LIN {X 0,Y 487.933,Z 756.497,A -85,B 0,C 180,E1 -6477.523,E2 -6477.523} C_VEL
LIN {X 0,Y 487.892,Z 757.524,A -85,B 0,C 180,E1 -6478.349,E2 -6478.349} C_VEL
LIN {X 0,Y 487.819,Z 758.415,A -85,B 0,C 180,E1 -6480,E2 -6480} C_VEL
LIN {X 0,Y 487.834,Z 758.228,A -85,B 0,C 180,E1 -6480.825,E2 -6480.825} C_VEL
LIN {X 0,Y 487.892,Z 757.637,A -85,B 0,C 180,E1 -6481.651,E2 -6481.651} C_VEL
LIN {X 0,Y 487.933,Z 756.658,A -85,B 0,C 180,E1 -6482.477,E2 -6482.477} C_VEL
LIN {X 0,Y 487.977,Z 755.262,A -85,B 0,C 180,E1 -6483.303,E2 -6483.303} C_VEL
LIN {X 0,Y 487.984,Z 752.337,A -85,B 0,C 180,E1 -6484.543,E2 -6484.543} C_VEL
LIN {X 0,Y 488.159,Z 747.294,A -85,B 0,C 180,E1 -6486.059,E2 -6486.059} C_VEL
LIN {X 0,Y 488.271,Z 741.184,A -85,B 0,C 180,E1 -6487.443,E2 -6487.443} C_VEL
LIN {X 0,Y 488.524,Z 734.149,A -85,B 0,C 180,E1 -6488.688,E2 -6488.688} C_VEL
LIN {X 0,Y 488.845,Z 725.387,A -85,B 0,C 180,E1 -6489.934,E2 -6489.934} C_VEL
LIN {X 0,Y 489.125,Z 716.359,A -85,B 0,C 180,E1 -6490.975,E2 -6490.975} C_VEL
LIN {X 0,Y 489.537,Z 706.321,A -85,B 0,C 180,E1 -6491.91,E2 -6491.91} C_VEL
LIN {X 0,Y 489.887,Z 695.409,A -85,B 0,C 180,E1 -6492.732,E2 -6492.732} C_VEL
LIN {X 0,Y 490.166,Z 683.839,A -85,B 0,C 180,E1 -6493.421,E2 -6493.421} C_VEL
LIN {X 0,Y 490.537,Z 670.88,A -85,B 0,C 180,E1 -6493.991,E2 -6493.991} C_VEL
LIN {X 0,Y 490.801,Z 658.232,A -85,B 0,C 180,E1 -6494.38,E2 -6494.38} C_VEL
LIN {X 0,Y 490.962,Z 638.871,A -85,B 0,C 180,E1 -6494.72,E2 -6494.72} C_VEL
LIN {X 0,Y 491.66,Z 557.51,A -85,B 0,C 180,E1 -6496.021,E2 -6496.021} C_VEL
LIN {X 0,Y 489.823,Z 546.055,A -85,B 0,C 180,E1 -6496.292,E2 -6496.292} C_VEL
LIN {X 0,Y 490.318,Z 525.468,A -85,B 0,C 180,E1 -6499.249,E2 -6499.249} C_VEL
LIN {X 0,Y 490.759,Z 505.581,A -85,B 0,C 180,E1 -6502.081,E2 -6502.081} C_VEL
LIN {X 0,Y 491.164,Z 488.188,A -85,B 0,C 180,E1 -6504.517,E2 -6504.517} C_VEL
LIN {X 0,Y 490.28,Z 481.713,A -85,B 0,C 180,E1 -6505.47,E2 -6505.47} C_VEL
LIN {X 0,Y 488.805,Z 474.727,A -85,B 0,C 180,E1 -6506.545,E2 -6506.545} C_VEL
LIN {X 0,Y 488.726,Z 474.734,A -85,B 0,C 180,E1 -6509.27,E2 -6509.27} C_VEL
LIN {X 0,Y 488.705,Z 474.737,A -85,B 0,C 180,E1 -6512.147,E2 -6512.147} C_VEL
LIN {X 0,Y 488.72,Z 474.734,A -85,B 0,C 180,E1 -6515.115,E2 -6515.115} C_VEL
LIN {X 0,Y 488.683,Z 474.738,A -85,B 0,C 180,E1 -6518.2,E2 -6518.2} C_VEL
LIN {X 0,Y 488.72,Z 474.734,A -85,B 0,C 180,E1 -6520.345,E2 -6520.345} C_VEL
LIN {X 0,Y 488.688,Z 474.733,A -85,B 0,C 180,E1 -6523.654,E2 -6523.654} C_VEL
LIN {X 0,Y 488.695,Z 474.738,A -85,B 0,C 180,E1 -6526.346,E2 -6526.346} C_VEL
LIN {X 0,Y 488.721,Z 474.734,A -85,B 0,C 180,E1 -6528.586,E2 -6528.586} C_VEL
LIN {X 0,Y 488.682,Z 474.736,A -85,B 0,C 180,E1 -6531.8,E2 -6531.8} C_VEL
LIN {X 0,Y 488.73,Z 474.73,A -85,B 0,C 180,E1 -6535.052,E2 -6535.052} C_VEL
LIN {X 0,Y 488.709,Z 474.735,A -85,B 0,C 180,E1 -6538.045,E2 -6538.045} C_VEL
LIN {X 0,Y 488.735,Z 474.733,A -85,B 0,C 180,E1 -6540.73,E2 -6540.73} C_VEL
LIN {X 0,Y 488.818,Z 474.835,A -85,B 0,C 180,E1 -6543.323,E2 -6543.323} C_VEL
LIN {X 0,Y 492.279,Z 490.053,A -85,B 0,C 180,E1 -6545.701,E2 -6545.701} C_VEL
LIN {X 0,Y 491.607,Z 506.366,A -85,B 0,C 180,E1 -6547.959,E2 -6547.959} C_VEL
LIN {X 0,Y 490.829,Z 524.604,A -85,B 0,C 180,E1 -6550.446,E2 -6550.446} C_VEL
LIN {X 0,Y 493.202,Z 539.821,A -85,B 0,C 180,E1 -6550.788,E2 -6550.788} C_VEL
LIN {X 0,Y 491.994,Z 662.426,A -85,B 0,C 180,E1 -6552.691,E2 -6552.691} C_VEL
LIN {X 0,Y 491.67,Z 676.703,A -85,B 0,C 180,E1 -6553.076,E2 -6553.076} C_VEL
LIN {X 0,Y 491.321,Z 691.164,A -85,B 0,C 180,E1 -6553.649,E2 -6553.649} C_VEL
LIN {X 0,Y 490.845,Z 703.923,A -85,B 0,C 180,E1 -6554.32,E2 -6554.32} C_VEL
LIN {X 0,Y 490.282,Z 716.464,A -85,B 0,C 180,E1 -6555.153,E2 -6555.153} C_VEL
LIN {X 0,Y 489.827,Z 727.924,A -85,B 0,C 180,E1 -6556.094,E2 -6556.094} C_VEL
LIN {X 0,Y 489.367,Z 738.441,A -85,B 0,C 180,E1 -6557.138,E2 -6557.138} C_VEL
LIN {X 0,Y 488.945,Z 748.885,A -85,B 0,C 180,E1 -6558.391,E2 -6558.391} C_VEL
LIN {X 0,Y 488.603,Z 757.487,A -85,B 0,C 180,E1 -6559.642,E2 -6559.642} C_VEL
LIN {X 0,Y 488.314,Z 765.679,A -85,B 0,C 180,E1 -6561.1,E2 -6561.1} C_VEL
LIN {X 0,Y 488.084,Z 772.266,A -85,B 0,C 180,E1 -6562.554,E2 -6562.554} C_VEL
LIN {X 0,Y 488.017,Z 776.821,A -85,B 0,C 180,E1 -6563.797,E2 -6563.797} C_VEL
LIN {X 0,Y 487.962,Z 780.398,A -85,B 0,C 180,E1 -6565.043,E2 -6565.043} C_VEL
LIN {X 0,Y 487.955,Z 783.88,A -85,B 0,C 180,E1 -6566.697,E2 -6566.697} C_VEL
LIN {X 0,Y 487.887,Z 785.935,A -85,B 0,C 180,E1 -6568.349,E2 -6568.349} C_VEL
LIN {X 0,Y 487.817,Z 786.61,A -85,B 0,C 180,E1 -6570,E2 -6570} C_VEL
LIN {X 0,Y 487.887,Z 785.914,A -85,B 0,C 180,E1 -6571.651,E2 -6571.651} C_VEL
LIN {X 0,Y 487.955,Z 783.837,A -85,B 0,C 180,E1 -6573.303,E2 -6573.303} C_VEL
LIN {X 0,Y 487.962,Z 780.328,A -85,B 0,C 180,E1 -6574.958,E2 -6574.958} C_VEL
LIN {X 0,Y 488.027,Z 775.834,A -85,B 0,C 180,E1 -6576.456,E2 -6576.456} C_VEL
LIN {X 0,Y 488.151,Z 770.373,A -85,B 0,C 180,E1 -6577.861,E2 -6577.861} C_VEL
LIN {X 0,Y 488.396,Z 763.274,A -85,B 0,C 180,E1 -6579.317,E2 -6579.317} C_VEL
LIN {X 0,Y 488.709,Z 754.438,A -85,B 0,C 180,E1 -6580.775,E2 -6580.775} C_VEL
LIN {X 0,Y 489.084,Z 744.365,A -85,B 0,C 180,E1 -6582.128,E2 -6582.128} C_VEL
LIN {X 0,Y 489.532,Z 732.81,A -85,B 0,C 180,E1 -6583.385,E2 -6583.385} C_VEL
LIN {X 0,Y 490.01,Z 721.006,A -85,B 0,C 180,E1 -6584.43,E2 -6584.43} C_VEL
LIN {X 0,Y 490.577,Z 707.861,A -85,B 0,C 180,E1 -6585.369,E2 -6585.369} C_VEL
LIN {X 0,Y 491.05,Z 694.161,A -85,B 0,C 180,E1 -6586.139,E2 -6586.139} C_VEL
LIN {X 0,Y 491.481,Z 679.477,A -85,B 0,C 180,E1 -6586.752,E2 -6586.752} C_VEL
LIN {X 0,Y 491.806,Z 666.25,A -85,B 0,C 180,E1 -6587.142,E2 -6587.142} C_VEL
LIN {X 0,Y 492.03,Z 648.794,A -85,B 0,C 180,E1 -6587.455,E2 -6587.455} C_VEL
LIN {X 0,Y 493.022,Z 539.589,A -85,B 0,C 180,E1 -6589.157,E2 -6589.157} C_VEL
LIN {X 0,Y 490.811,Z 525.078,A -85,B 0,C 180,E1 -6589.491,E2 -6589.491} C_VEL
LIN {X 0,Y 492.007,Z 500.536,A -85,B 0,C 180,E1 -6592.908,E2 -6592.908} C_VEL
LIN {X 0,Y 492.543,Z 491.86,A -85,B 0,C 180,E1 -6594.152,E2 -6594.152} C_VEL
LIN {X 0,Y 491.719,Z 486.921,A -85,B 0,C 180,E1 -6594.938,E2 -6594.938} C_VEL
LIN {X 0,Y 489.179,Z 476.31,A -85,B 0,C 180,E1 -6596.751,E2 -6596.751} C_VEL
LIN {X 0,Y 488.79,Z 474.727,A -85,B 0,C 180,E1 -6597.058,E2 -6597.058} C_VEL
LIN {X 0,Y 488.713,Z 474.736,A -85,B 0,C 180,E1 -6600.363,E2 -6600.363} C_VEL
LIN {X 0,Y 488.737,Z 474.734,A -85,B 0,C 180,E1 -6603.484,E2 -6603.484} C_VEL
LIN {X 0,Y 488.684,Z 474.737,A -85,B 0,C 180,E1 -6606.355,E2 -6606.355} C_VEL
LIN {X 0,Y 488.703,Z 474.738,A -85,B 0,C 180,E1 -6609.254,E2 -6609.254} C_VEL
LIN {X 0,Y 488.726,Z 474.733,A -85,B 0,C 180,E1 -6611.602,E2 -6611.602} C_VEL
LIN {X 0,Y 488.715,Z 474.734,A -85,B 0,C 180,E1 -6614.801,E2 -6614.801} C_VEL
LIN {X 0,Y 488.694,Z 474.736,A -85,B 0,C 180,E1 -6617.475,E2 -6617.475} C_VEL
LIN {X 0,Y 488.736,Z 474.73,A -85,B 0,C 180,E1 -6619.677,E2 -6619.677} C_VEL
LIN {X 0,Y 488.683,Z 474.741,A -85,B 0,C 180,E1 -6622.841,E2 -6622.841} C_VEL
LIN {X 0,Y 488.736,Z 474.731,A -85,B 0,C 180,E1 -6625.888,E2 -6625.888} C_VEL
LIN {X 0,Y 488.697,Z 474.74,A -85,B 0,C 180,E1 -6628.821,E2 -6628.821} C_VEL
LIN {X 0,Y 488.749,Z 474.735,A -85,B 0,C 180,E1 -6631.671,E2 -6631.671} C_VEL
LIN {X 0,Y 488.806,Z 474.846,A -85,B 0,C 180,E1 -6633.646,E2 -6633.646} C_VEL
LIN {X 0,Y 491.471,Z 486.878,A -85,B 0,C 180,E1 -6635.912,E2 -6635.912} C_VEL
LIN {X 0,Y 491.925,Z 491.046,A -85,B 0,C 180,E1 -6636.643,E2 -6636.643} C_VEL
LIN {X 0,Y 490.778,Z 512.524,A -85,B 0,C 180,E1 -6640.117,E2 -6640.117} C_VEL
LIN {X 0,Y 490.085,Z 530.15,A -85,B 0,C 180,E1 -6642.904,E2 -6642.904} C_VEL
LIN {X 0,Y 489.754,Z 540.863,A -85,B 0,C 180,E1 -6644.578,E2 -6644.578} C_VEL
LIN {X 0,Y 492.036,Z 554.998,A -85,B 0,C 180,E1 -6644.916,E2 -6644.916} C_VEL
LIN {X 0,Y 490.94,Z 653.001,A -85,B 0,C 180,E1 -6646.575,E2 -6646.575} C_VEL
LIN {X 0,Y 490.687,Z 666.595,A -85,B 0,C 180,E1 -6646.98,E2 -6646.98} C_VEL
LIN {X 0,Y 490.427,Z 679.005,A -85,B 0,C 180,E1 -6647.52,E2 -6647.52} C_VEL
LIN {X 0,Y 490.086,Z 690.877,A -85,B 0,C 180,E1 -6648.209,E2 -6648.209} C_VEL
LIN {X 0,Y 489.611,Z 702.158,A -85,B 0,C 180,E1 -6649.036,E2 -6649.036} C_VEL
LIN {X 0,Y 489.215,Z 712.339,A -85,B 0,C 180,E1 -6649.969,E2 -6649.969} C_VEL
LIN {X 0,Y 488.877,Z 722.337,A -85,B 0,C 180,E1 -6651.11,E2 -6651.11} C_VEL
LIN {X 0,Y 488.51,Z 731.141,A -85,B 0,C 180,E1 -6652.353,E2 -6652.353} C_VEL
LIN {X 0,Y 488.403,Z 738.144,A -85,B 0,C 180,E1 -6653.597,E2 -6653.597} C_VEL
LIN {X 0,Y 488.04,Z 744.561,A -85,B 0,C 180,E1 -6655.043,E2 -6655.043} C_VEL
LIN {X 0,Y 488.059,Z 748.762,A -85,B 0,C 180,E1 -6656.285,E2 -6656.285} C_VEL
LIN {X 0,Y 487.993,Z 751.895,A -85,B 0,C 180,E1 -6657.524,E2 -6657.524} C_VEL
LIN {X 0,Y 487.899,Z 753.453,A -85,B 0,C 180,E1 -6658.349,E2 -6658.349} C_VEL
LIN {X 0,Y 487.835,Z 754.563,A -85,B 0,C 180,E1 -6659.175,E2 -6659.175} C_VEL
LIN {X 0,Y 487.834,Z 755.556,A -85,B 0,C 180,E1 -6660.825,E2 -6660.825} C_VEL
LIN {X 0,Y 487.892,Z 755.467,A -85,B 0,C 180,E1 -6661.651,E2 -6661.651} C_VEL
LIN {X 0,Y 487.93,Z 754.951,A -85,B 0,C 180,E1 -6662.477,E2 -6662.477} C_VEL
LIN {X 0,Y 487.963,Z 754.02,A -85,B 0,C 180,E1 -6663.303,E2 -6663.303} C_VEL
LIN {X 0,Y 487.965,Z 752.694,A -85,B 0,C 180,E1 -6664.13,E2 -6664.13} C_VEL
LIN {X 0,Y 488.041,Z 749.887,A -85,B 0,C 180,E1 -6665.371,E2 -6665.371} C_VEL
LIN {X 0,Y 488.076,Z 745.518,A -85,B 0,C 180,E1 -6666.758,E2 -6666.758} C_VEL
LIN {X 0,Y 488.19,Z 741.056,A -85,B 0,C 180,E1 -6667.861,E2 -6667.861} C_VEL
LIN {X 0,Y 488.424,Z 734.771,A -85,B 0,C 180,E1 -6669.107,E2 -6669.107} C_VEL
LIN {X 0,Y 488.662,Z 726.91,A -85,B 0,C 180,E1 -6670.357,E2 -6670.357} C_VEL
LIN {X 0,Y 489.115,Z 717.067,A -85,B 0,C 180,E1 -6671.605,E2 -6671.605} C_VEL
LIN {X 0,Y 489.305,Z 709.051,A -85,B 0,C 180,E1 -6672.442,E2 -6672.442} C_VEL
LIN {X 0,Y 489.761,Z 698.135,A -85,B 0,C 180,E1 -6673.379,E2 -6673.379} C_VEL
LIN {X 0,Y 490.147,Z 687.485,A -85,B 0,C 180,E1 -6674.108,E2 -6674.108} C_VEL
LIN {X 0,Y 490.517,Z 675.852,A -85,B 0,C 180,E1 -6674.733,E2 -6674.733} C_VEL
LIN {X 0,Y 490.726,Z 662.767,A -85,B 0,C 180,E1 -6675.258,E2 -6675.258} C_VEL
LIN {X 0,Y 491.027,Z 650.035,A -85,B 0,C 180,E1 -6675.594,E2 -6675.594} C_VEL
LIN {X 0,Y 491.814,Z 554.672,A -85,B 0,C 180,E1 -6677.124,E2 -6677.124} C_VEL
LIN {X 0,Y 489.666,Z 541.039,A -85,B 0,C 180,E1 -6677.453,E2 -6677.453} C_VEL
LIN {X 0,Y 490.231,Z 525.254,A -85,B 0,C 180,E1 -6679.906,E2 -6679.906} C_VEL
LIN {X 0,Y 490.932,Z 507.268,A -85,B 0,C 180,E1 -6682.738,E2 -6682.738} C_VEL
LIN {X 0,Y 491.668,Z 490.617,A -85,B 0,C 180,E1 -6685.393,E2 -6685.393} C_VEL
LIN {X 0,Y 491.279,Z 486.187,A -85,B 0,C 180,E1 -6686.137,E2 -6686.137} C_VEL
LIN {X 0,Y 488.781,Z 474.728,A -85,B 0,C 180,E1 -6688.21,E2 -6688.21} C_VEL
LIN {X 0,Y 488.695,Z 474.737,A -85,B 0,C 180,E1 -6691.18,E2 -6691.18} C_VEL
LIN {X 0,Y 488.736,Z 474.73,A -85,B 0,C 180,E1 -6694.112,E2 -6694.112} C_VEL
LIN {X 0,Y 488.683,Z 474.735,A -85,B 0,C 180,E1 -6697.159,E2 -6697.159} C_VEL
LIN {X 0,Y 488.721,Z 474.728,A -85,B 0,C 180,E1 -6700.344,E2 -6700.344} C_VEL
LIN {X 0,Y 488.687,Z 474.74,A -85,B 0,C 180,E1 -6703.654,E2 -6703.654} C_VEL
LIN {X 0,Y 488.694,Z 474.733,A -85,B 0,C 180,E1 -6705.382,E2 -6705.382} C_VEL
LIN {X 0,Y 488.017,Z 474.819,A -85,B 0,C 180,E1 -6706.07,E2 -6706.07} C_VEL
LIN {X 0,Y 485.167,Z 475.174,A -85,B 0,C 180,E1 -6707.187,E2 -6707.187} C_VEL
LIN {X 0,Y 482.767,Z 475.472,A -85,B 0,C 180,E1 -6708.087,E2 -6708.087} C_VEL
LIN {X 0,Y 481.74,Z 475.598,A -85,B 0,C 180,E1 -6708.782,E2 -6708.782} C_VEL
LIN {X 0,Y 481.658,Z 475.609,A -85,B 0,C 180,E1 -6709.018,E2 -6709.018} C_VEL
LIN {X 0,Y 481.657,Z 475.611,A -85,B 0,C 180,E1 -6711.993,E2 -6711.993} C_VEL
LIN {X 0,Y 481.69,Z 475.609,A -85,B 0,C 180,E1 -6715.318,E2 -6715.318} C_VEL
LIN {X 0,Y 481.647,Z 475.609,A -85,B 0,C 180,E1 -6718.311,E2 -6718.311} C_VEL
LIN {X 0,Y 481.702,Z 475.606,A -85,B 0,C 180,E1 -6721.218,E2 -6721.218} C_VEL
LIN {X 0,Y 481.703,Z 475.604,A -85,B 0,C 180,E1 -6724.043,E2 -6724.043} C_VEL
LIN {X 0,Y 481.676,Z 475.606,A -85,B 0,C 180,E1 -6726.812,E2 -6726.812} C_VEL
LIN {X 0,Y 481.699,Z 475.611,A -85,B 0,C 180,E1 -6729.503,E2 -6729.503} C_VEL
LIN {X 0,Y 481.709,Z 475.602,A -85,B 0,C 180,E1 -6732.158,E2 -6732.158} C_VEL
LIN {X 0,Y 481.746,Z 475.597,A -85,B 0,C 180,E1 -6734.776,E2 -6734.776} C_VEL
LIN {X 0,Y 481.753,Z 475.596,A -85,B 0,C 180,E1 -6738.215,E2 -6738.215} C_VEL
LIN {X 0,Y 481.766,Z 475.601,A -85,B 0,C 180,E1 -6741.612,E2 -6741.612} C_VEL
LIN {X 0,Y 481.818,Z 475.589,A -85,B 0,C 180,E1 -6744.14,E2 -6744.14} C_VEL
LIN {X 0,Y 481.931,Z 475.582,A -85,B 0,C 180,E1 -6747.493,E2 -6747.493} C_VEL
LIN {X 0,Y 481.908,Z 475.578,A -85,B 0,C 180,E1 -6750.836,E2 -6750.836} C_VEL
LIN {X 0,Y 481.931,Z 475.574,A -85,B 0,C 180,E1 -6752.507,E2 -6752.507} C_VEL
LIN {X 0,Y 481.811,Z 475.591,A -85,B 0,C 180,E1 -6755.86,E2 -6755.86} C_VEL
LIN {X 0,Y 481.765,Z 475.594,A -85,B 0,C 180,E1 -6758.388,E2 -6758.388} C_VEL
LIN {X 0,Y 481.753,Z 475.599,A -85,B 0,C 180,E1 -6761.785,E2 -6761.785} C_VEL
LIN {X 0,Y 481.745,Z 475.603,A -85,B 0,C 180,E1 -6765.224,E2 -6765.224} C_VEL
LIN {X 0,Y 481.714,Z 475.602,A -85,B 0,C 180,E1 -6768.722,E2 -6768.722} C_VEL
LIN {X 0,Y 481.65,Z 475.617,A -85,B 0,C 180,E1 -6771.395,E2 -6771.395} C_VEL
LIN {X 0,Y 481.679,Z 475.605,A -85,B 0,C 180,E1 -6774.113,E2 -6774.113} C_VEL
LIN {X 0,Y 481.749,Z 475.602,A -85,B 0,C 180,E1 -6777.139,E2 -6777.139} C_VEL
LIN {X 0,Y 481.68,Z 475.608,A -85,B 0,C 180,E1 -6779.741,E2 -6779.741} C_VEL
LIN {X 0,Y 481.673,Z 475.607,A -85,B 0,C 180,E1 -6782.674,E2 -6782.674} C_VEL
LIN {X 0,Y 481.638,Z 475.614,A -85,B 0,C 180,E1 -6785.71,E2 -6785.71} C_VEL
LIN {X 0,Y 481.673,Z 475.608,A -85,B 0,C 180,E1 -6788.859,E2 -6788.859} C_VEL
LIN {X 0,Y 481.665,Z 475.608,A -85,B 0,C 180,E1 -6791.914,E2 -6791.914} C_VEL
LIN {X 0,Y 481.662,Z 475.607,A -85,B 0,C 180,E1 -6794.457,E2 -6794.457} C_VEL
LIN {X 0,Y 481.649,Z 475.611,A -85,B 0,C 180,E1 -6797.839,E2 -6797.839} C_VEL
LIN {X 0,Y 481.683,Z 475.606,A -85,B 0,C 180,E1 -6800.651,E2 -6800.651} C_VEL
LIN {X 0,Y 481.63,Z 475.619,A -85,B 0,C 180,E1 -6803.376,E2 -6803.376} C_VEL
LIN {X 0,Y 481.712,Z 475.601,A -85,B 0,C 180,E1 -6806.33,E2 -6806.33} C_VEL
LIN {X 0,Y 481.653,Z 475.614,A -85,B 0,C 180,E1 -6809.417,E2 -6809.417} C_VEL
LIN {X 0,Y 481.703,Z 475.604,A -85,B 0,C 180,E1 -6812.168,E2 -6812.168} C_VEL
LIN {X 0,Y 481.764,Z 475.705,A -85,B 0,C 180,E1 -6812.99,E2 -6812.99} C_VEL
LIN {X 0,Y 484.474,Z 488.91,A -85,B 0,C 180,E1 -6815.122,E2 -6815.122} C_VEL
LIN {X 0,Y 484.028,Z 507.022,A -85,B 0,C 180,E1 -6817.82,E2 -6817.82} C_VEL
LIN {X 0,Y 483.345,Z 528.893,A -85,B 0,C 180,E1 -6821.071,E2 -6821.071} C_VEL
LIN {X 0,Y 482.826,Z 545.753,A -85,B 0,C 180,E1 -6823.569,E2 -6823.569} C_VEL
LIN {X 0,Y 484.843,Z 559.043,A -85,B 0,C 180,E1 -6823.861,E2 -6823.861} C_VEL
LIN {X 0,Y 484.014,Z 655.064,A -85,B 0,C 180,E1 -6825.414,E2 -6825.414} C_VEL
LIN {X 0,Y 483.771,Z 667.39,A -85,B 0,C 180,E1 -6825.756,E2 -6825.756} C_VEL
LIN {X 0,Y 483.396,Z 680.173,A -85,B 0,C 180,E1 -6826.281,E2 -6826.281} C_VEL
LIN {X 0,Y 483.021,Z 692.411,A -85,B 0,C 180,E1 -6826.967,E2 -6826.967} C_VEL
LIN {X 0,Y 482.77,Z 702.747,A -85,B 0,C 180,E1 -6827.707,E2 -6827.707} C_VEL
LIN {X 0,Y 482.311,Z 713.398,A -85,B 0,C 180,E1 -6828.655,E2 -6828.655} C_VEL
LIN {X 0,Y 481.928,Z 722.972,A -85,B 0,C 180,E1 -6829.709,E2 -6829.709} C_VEL
LIN {X 0,Y 481.593,Z 730.844,A -85,B 0,C 180,E1 -6830.763,E2 -6830.763} C_VEL
LIN {X 0,Y 481.309,Z 738.549,A -85,B 0,C 180,E1 -6832.026,E2 -6832.026} C_VEL
LIN {X 0,Y 481.106,Z 745.101,A -85,B 0,C 180,E1 -6833.388,E2 -6833.388} C_VEL
LIN {X 0,Y 481.02,Z 749.544,A -85,B 0,C 180,E1 -6834.55,E2 -6834.55} C_VEL
LIN {X 0,Y 480.933,Z 753.273,A -85,B 0,C 180,E1 -6835.81,E2 -6835.81} C_VEL
LIN {X 0,Y 480.907,Z 755.19,A -85,B 0,C 180,E1 -6836.649,E2 -6836.649} C_VEL
LIN {X 0,Y 480.846,Z 756.676,A -85,B 0,C 180,E1 -6837.487,E2 -6837.487} C_VEL
LIN {X 0,Y 480.823,Z 757.708,A -85,B 0,C 180,E1 -6838.325,E2 -6838.325} C_VEL
LIN {X 0,Y 480.743,Z 758.607,A -85,B 0,C 180,E1 -6840,E2 -6840} C_VEL
LIN {X 0,Y 480.76,Z 758.42,A -85,B 0,C 180,E1 -6840.838,E2 -6840.838} C_VEL
LIN {X 0,Y 480.823,Z 757.826,A -85,B 0,C 180,E1 -6841.675,E2 -6841.675} C_VEL
LIN {X 0,Y 480.846,Z 756.843,A -85,B 0,C 180,E1 -6842.513,E2 -6842.513} C_VEL
LIN {X 0,Y 480.906,Z 755.438,A -85,B 0,C 180,E1 -6843.351,E2 -6843.351} C_VEL
LIN {X 0,Y 480.89,Z 752.498,A -85,B 0,C 180,E1 -6844.61,E2 -6844.61} C_VEL
LIN {X 0,Y 481.081,Z 748.486,A -85,B 0,C 180,E1 -6845.869,E2 -6845.869} C_VEL
LIN {X 0,Y 481.187,Z 742.289,A -85,B 0,C 180,E1 -6847.342,E2 -6847.342} C_VEL
LIN {X 0,Y 481.442,Z 735.513,A -85,B 0,C 180,E1 -6848.605,E2 -6848.605} C_VEL
LIN {X 0,Y 481.749,Z 727.002,A -85,B 0,C 180,E1 -6849.87,E2 -6849.87} C_VEL
LIN {X 0,Y 482.047,Z 718.272,A -85,B 0,C 180,E1 -6850.926,E2 -6850.926} C_VEL
LIN {X 0,Y 482.473,Z 708.689,A -85,B 0,C 180,E1 -6851.874,E2 -6851.874} C_VEL
LIN {X 0,Y 482.847,Z 698.303,A -85,B 0,C 180,E1 -6852.707,E2 -6852.707} C_VEL
LIN {X 0,Y 483.167,Z 686.482,A -85,B 0,C 180,E1 -6853.458,E2 -6853.458} C_VEL
LIN {X 0,Y 483.51,Z 674.547,A -85,B 0,C 180,E1 -6854.038,E2 -6854.038} C_VEL
LIN {X 0,Y 483.84,Z 661.492,A -85,B 0,C 180,E1 -6854.484,E2 -6854.484} C_VEL
LIN {X 0,Y 484.048,Z 647.823,A -85,B 0,C 180,E1 -6854.773,E2 -6854.773} C_VEL
LIN {X 0,Y 484.774,Z 557.802,A -85,B 0,C 180,E1 -6856.253,E2 -6856.253} C_VEL
LIN {X 0,Y 482.936,Z 546.23,A -85,B 0,C 180,E1 -6856.547,E2 -6856.547} C_VEL
LIN {X 0,Y 483.514,Z 524.071,A -85,B 0,C 180,E1 -6859.752,E2 -6859.752} C_VEL
LIN {X 0,Y 483.99,Z 503.956,A -85,B 0,C 180,E1 -6862.632,E2 -6862.632} C_VEL
LIN {X 0,Y 484.322,Z 489.61,A -85,B 0,C 180,E1 -6864.657,E2 -6864.657} C_VEL
LIN {X 0,Y 483.025,Z 481.443,A -85,B 0,C 180,E1 -6865.881,E2 -6865.881} C_VEL
LIN {X 0,Y 481.744,Z 475.607,A -85,B 0,C 180,E1 -6866.8,E2 -6866.8} C_VEL
LIN {X 0,Y 481.682,Z 475.61,A -85,B 0,C 180,E1 -6869.741,E2 -6869.741} C_VEL
LIN {X 0,Y 481.674,Z 475.616,A -85,B 0,C 180,E1 -6872.674,E2 -6872.674} C_VEL
LIN {X 0,Y 481.639,Z 475.613,A -85,B 0,C 180,E1 -6875.709,E2 -6875.709} C_VEL
LIN {X 0,Y 481.674,Z 475.612,A -85,B 0,C 180,E1 -6878.859,E2 -6878.859} C_VEL
LIN {X 0,Y 481.654,Z 475.611,A -85,B 0,C 180,E1 -6881.913,E2 -6881.913} C_VEL
LIN {X 0,Y 481.662,Z 475.614,A -85,B 0,C 180,E1 -6884.457,E2 -6884.457} C_VEL
LIN {X 0,Y 481.656,Z 475.61,A -85,B 0,C 180,E1 -6887.84,E2 -6887.84} C_VEL
LIN {X 0,Y 481.682,Z 475.61,A -85,B 0,C 180,E1 -6890.651,E2 -6890.651} C_VEL
LIN {X 0,Y 481.633,Z 475.613,A -85,B 0,C 180,E1 -6893.375,E2 -6893.375} C_VEL
LIN {X 0,Y 481.712,Z 475.607,A -85,B 0,C 180,E1 -6896.33,E2 -6896.33} C_VEL
LIN {X 0,Y 481.661,Z 475.611,A -85,B 0,C 180,E1 -6899.416,E2 -6899.416} C_VEL
LIN {X 0,Y 481.703,Z 475.61,A -85,B 0,C 180,E1 -6902.168,E2 -6902.168} C_VEL
LIN {X 0,Y 481.769,Z 475.694,A -85,B 0,C 180,E1 -6903.031,E2 -6903.031} C_VEL
LIN {X 0,Y 485.46,Z 491.804,A -85,B 0,C 180,E1 -6905.595,E2 -6905.595} C_VEL
LIN {X 0,Y 484.628,Z 509.543,A -85,B 0,C 180,E1 -6908.081,E2 -6908.081} C_VEL
LIN {X 0,Y 483.944,Z 524.654,A -85,B 0,C 180,E1 -6910.17,E2 -6910.17} C_VEL
LIN {X 0,Y 486.475,Z 540.36,A -85,B 0,C 180,E1 -6910.538,E2 -6910.538} C_VEL
LIN {X 0,Y 485.145,Z 662.579,A -85,B 0,C 180,E1 -6912.48,E2 -6912.48} C_VEL
LIN {X 0,Y 484.791,Z 676.893,A -85,B 0,C 180,E1 -6912.874,E2 -6912.874} C_VEL
LIN {X 0,Y 484.45,Z 690.472,A -85,B 0,C 180,E1 -6913.419,E2 -6913.419} C_VEL
LIN {X 0,Y 483.966,Z 703.223,A -85,B 0,C 180,E1 -6914.092,E2 -6914.092} C_VEL
LIN {X 0,Y 483.345,Z 715.867,A -85,B 0,C 180,E1 -6914.935,E2 -6914.935} C_VEL
LIN {X 0,Y 482.826,Z 727.404,A -85,B 0,C 180,E1 -6915.888,E2 -6915.888} C_VEL
LIN {X 0,Y 482.367,Z 737.987,A -85,B 0,C 180,E1 -6916.948,E2 -6916.948} C_VEL
LIN {X 0,Y 481.944,Z 748.494,A -85,B 0,C 180,E1 -6918.22,E2 -6918.22} C_VEL
LIN {X 0,Y 481.571,Z 757.138,A -85,B 0,C 180,E1 -6919.489,E2 -6919.489} C_VEL
LIN {X 0,Y 481.263,Z 765.37,A -85,B 0,C 180,E1 -6920.968,E2 -6920.968} C_VEL
LIN {X 0,Y 481.009,Z 771.984,A -85,B 0,C 180,E1 -6922.444,E2 -6922.444} C_VEL
LIN {X 0,Y 480.963,Z 775.975,A -85,B 0,C 180,E1 -6923.535,E2 -6923.535} C_VEL
LIN {X 0,Y 480.893,Z 780.15,A -85,B 0,C 180,E1 -6924.969,E2 -6924.969} C_VEL
LIN {X 0,Y 480.879,Z 783.645,A -85,B 0,C 180,E1 -6926.649,E2 -6926.649} C_VEL
LIN {X 0,Y 480.818,Z 785.709,A -85,B 0,C 180,E1 -6928.325,E2 -6928.325} C_VEL
LIN {X 0,Y 480.741,Z 786.386,A -85,B 0,C 180,E1 -6930,E2 -6930} C_VEL
LIN {X 0,Y 480.818,Z 785.682,A -85,B 0,C 180,E1 -6931.675,E2 -6931.675} C_VEL
LIN {X 0,Y 480.879,Z 783.591,A -85,B 0,C 180,E1 -6933.351,E2 -6933.351} C_VEL
LIN {X 0,Y 480.894,Z 780.057,A -85,B 0,C 180,E1 -6935.031,E2 -6935.031} C_VEL
LIN {X 0,Y 480.962,Z 774.969,A -85,B 0,C 180,E1 -6936.713,E2 -6936.713} C_VEL
LIN {X 0,Y 481.082,Z 770.038,A -85,B 0,C 180,E1 -6937.978,E2 -6937.978} C_VEL
LIN {X 0,Y 481.339,Z 762.894,A -85,B 0,C 180,E1 -6939.454,E2 -6939.454} C_VEL
LIN {X 0,Y 481.692,Z 754.009,A -85,B 0,C 180,E1 -6940.934,E2 -6940.934} C_VEL
LIN {X 0,Y 482.044,Z 744.639,A -85,B 0,C 180,E1 -6942.21,E2 -6942.21} C_VEL
LIN {X 0,Y 482.459,Z 734.347,A -85,B 0,C 180,E1 -6943.371,E2 -6943.371} C_VEL
LIN {X 0,Y 482.92,Z 722.94,A -85,B 0,C 180,E1 -6944.432,E2 -6944.432} C_VEL
LIN {X 0,Y 483.496,Z 710.262,A -85,B 0,C 180,E1 -6945.384,E2 -6945.384} C_VEL
LIN {X 0,Y 484.028,Z 696.945,A -85,B 0,C 180,E1 -6946.177,E2 -6946.177} C_VEL
LIN {X 0,Y 484.456,Z 683.366,A -85,B 0,C 180,E1 -6946.8,E2 -6946.8} C_VEL
LIN {X 0,Y 484.837,Z 669.561,A -85,B 0,C 180,E1 -6947.26,E2 -6947.26} C_VEL
LIN {X 0,Y 485.1,Z 656.216,A -85,B 0,C 180,E1 -6947.549,E2 -6947.549} C_VEL
LIN {X 0,Y 486.272,Z 542.803,A -85,B 0,C 180,E1 -6949.36,E2 -6949.36} C_VEL
LIN {X 0,Y 485.904,Z 537.671,A -85,B 0,C 180,E1 -6949.464,E2 -6949.464} C_VEL
LIN {X 0,Y 483.972,Z 525.311,A -85,B 0,C 180,E1 -6949.761,E2 -6949.761} C_VEL
LIN {X 0,Y 485.301,Z 500.827,A -85,B 0,C 180,E1 -6953.243,E2 -6953.243} C_VEL
LIN {X 0,Y 485.728,Z 492.563,A -85,B 0,C 180,E1 -6954.462,E2 -6954.462} C_VEL
LIN {X 0,Y 483.303,Z 481.664,A -85,B 0,C 180,E1 -6956.329,E2 -6956.329} C_VEL
LIN {X 0,Y 481.711,Z 475.61,A -85,B 0,C 180,E1 -6957.441,E2 -6957.441} C_VEL
LIN {X 0,Y 481.654,Z 475.615,A -85,B 0,C 180,E1 -6960.583,E2 -6960.583} C_VEL
LIN {X 0,Y 481.699,Z 475.61,A -85,B 0,C 180,E1 -6963.733,E2 -6963.733} C_VEL
LIN {X 0,Y 481.628,Z 475.617,A -85,B 0,C 180,E1 -6966.747,E2 -6966.747} C_VEL
LIN {X 0,Y 481.679,Z 475.61,A -85,B 0,C 180,E1 -6969.94,E2 -6969.94} C_VEL
LIN {X 0,Y 481.669,Z 475.613,A -85,B 0,C 180,E1 -6973.297,E2 -6973.297} C_VEL
LIN {X 0,Y 481.661,Z 475.612,A -85,B 0,C 180,E1 -6975.641,E2 -6975.641} C_VEL
LIN {X 0,Y 481.659,Z 475.615,A -85,B 0,C 180,E1 -6978.958,E2 -6978.958} C_VEL
LIN {X 0,Y 481.658,Z 475.612,A -85,B 0,C 180,E1 -6981.993,E2 -6981.993} C_VEL
LIN {X 0,Y 481.693,Z 475.61,A -85,B 0,C 180,E1 -6985.318,E2 -6985.318} C_VEL
LIN {X 0,Y 481.649,Z 475.616,A -85,B 0,C 180,E1 -6988.312,E2 -6988.312} C_VEL
LIN {X 0,Y 481.704,Z 475.614,A -85,B 0,C 180,E1 -6991.219,E2 -6991.219} C_VEL
LIN {X 0,Y 481.753,Z 475.722,A -85,B 0,C 180,E1 -6993.259,E2 -6993.259} C_VEL
LIN {X 0,Y 484.21,Z 486.33,A -85,B 0,C 180,E1 -6995.337,E2 -6995.337} C_VEL
LIN {X 0,Y 485.139,Z 491.5,A -85,B 0,C 180,E1 -6996.297,E2 -6996.297} C_VEL
LIN {X 0,Y 484.105,Z 510.182,A -85,B 0,C 180,E1 -6999.387,E2 -6999.387} C_VEL
LIN {X 0,Y 483.174,Z 530.422,A -85,B 0,C 180,E1 -7002.652,E2 -7002.652} C_VEL
LIN {X 0,Y 482.84,Z 540.843,A -85,B 0,C 180,E1 -7004.291,E2 -7004.291} C_VEL
LIN {X 0,Y 485.312,Z 555.99,A -85,B 0,C 180,E1 -7004.675,E2 -7004.675} C_VEL
LIN {X 0,Y 484.282,Z 639.622,A -85,B 0,C 180,E1 -7006.119,E2 -7006.119} C_VEL
LIN {X 0,Y 484.012,Z 655.637,A -85,B 0,C 180,E1 -7006.432,E2 -7006.432} C_VEL
LIN {X 0,Y 483.763,Z 668.415,A -85,B 0,C 180,E1 -7006.849,E2 -7006.849} C_VEL
LIN {X 0,Y 483.479,Z 680.503,A -85,B 0,C 180,E1 -7007.406,E2 -7007.406} C_VEL
LIN {X 0,Y 483.137,Z 691.104,A -85,B 0,C 180,E1 -7008.036,E2 -7008.036} C_VEL
LIN {X 0,Y 482.659,Z 702.37,A -85,B 0,C 180,E1 -7008.876,E2 -7008.876} C_VEL
LIN {X 0,Y 482.224,Z 712.544,A -85,B 0,C 180,E1 -7009.822,E2 -7009.822} C_VEL
LIN {X 0,Y 481.873,Z 722.544,A -85,B 0,C 180,E1 -7010.98,E2 -7010.98} C_VEL
LIN {X 0,Y 481.483,Z 731.352,A -85,B 0,C 180,E1 -7012.24,E2 -7012.24} C_VEL
LIN {X 0,Y 481.335,Z 738.105,A -85,B 0,C 180,E1 -7013.448,E2 -7013.448} C_VEL
LIN {X 0,Y 481.067,Z 743.162,A -85,B 0,C 180,E1 -7014.551,E2 -7014.551} C_VEL
LIN {X 0,Y 481.059,Z 747.749,A -85,B 0,C 180,E1 -7015.811,E2 -7015.811} C_VEL
LIN {X 0,Y 480.946,Z 750.164,A -85,B 0,C 180,E1 -7016.649,E2 -7016.649} C_VEL
LIN {X 0,Y 480.902,Z 752.141,A -85,B 0,C 180,E1 -7017.487,E2 -7017.487} C_VEL
LIN {X 0,Y 480.831,Z 753.699,A -85,B 0,C 180,E1 -7018.325,E2 -7018.325} C_VEL
LIN {X 0,Y 480.761,Z 754.803,A -85,B 0,C 180,E1 -7019.162,E2 -7019.162} C_VEL
LIN {X 0,Y 480.76,Z 755.785,A -85,B 0,C 180,E1 -7020.838,E2 -7020.838} C_VEL
LIN {X 0,Y 480.823,Z 755.687,A -85,B 0,C 180,E1 -7021.675,E2 -7021.675} C_VEL
LIN {X 0,Y 480.843,Z 755.156,A -85,B 0,C 180,E1 -7022.513,E2 -7022.513} C_VEL
LIN {X 0,Y 480.89,Z 754.213,A -85,B 0,C 180,E1 -7023.351,E2 -7023.351} C_VEL
LIN {X 0,Y 480.868,Z 752.872,A -85,B 0,C 180,E1 -7024.191,E2 -7024.191} C_VEL
LIN {X 0,Y 480.977,Z 750.036,A -85,B 0,C 180,E1 -7025.45,E2 -7025.45} C_VEL
LIN {X 0,Y 481.006,Z 745.954,A -85,B 0,C 180,E1 -7026.769,E2 -7026.769} C_VEL
LIN {X 0,Y 481.137,Z 741.13,A -85,B 0,C 180,E1 -7027.976,E2 -7027.976} C_VEL
LIN {X 0,Y 481.365,Z 734.799,A -85,B 0,C 180,E1 -7029.242,E2 -7029.242} C_VEL
LIN {X 0,Y 481.653,Z 726.873,A -85,B 0,C 180,E1 -7030.509,E2 -7030.509} C_VEL
LIN {X 0,Y 482.045,Z 718.774,A -85,B 0,C 180,E1 -7031.564,E2 -7031.564} C_VEL
LIN {X 0,Y 482.265,Z 710.422,A -85,B 0,C 180,E1 -7032.475,E2 -7032.475} C_VEL
LIN {X 0,Y 482.767,Z 699.213,A -85,B 0,C 180,E1 -7033.469,E2 -7033.469} C_VEL
LIN {X 0,Y 483.186,Z 688.834,A -85,B 0,C 180,E1 -7034.208,E2 -7034.208} C_VEL
LIN {X 0,Y 483.572,Z 677.618,A -85,B 0,C 180,E1 -7034.842,E2 -7034.842} C_VEL
LIN {X 0,Y 483.831,Z 664.366,A -85,B 0,C 180,E1 -7035.4,E2 -7035.4} C_VEL
LIN {X 0,Y 484.131,Z 651.418,A -85,B 0,C 180,E1 -7035.768,E2 -7035.768} C_VEL
LIN {X 0,Y 485.117,Z 556.06,A -85,B 0,C 180,E1 -7037.338,E2 -7037.338} C_VEL
LIN {X 0,Y 482.73,Z 541.086,A -85,B 0,C 180,E1 -7037.689,E2 -7037.689} C_VEL
LIN {X 0,Y 483.329,Z 525.152,A -85,B 0,C 180,E1 -7040.203,E2 -7040.203} C_VEL
LIN {X 0,Y 484.069,Z 507.134,A -85,B 0,C 180,E1 -7043.079,E2 -7043.079} C_VEL
LIN {X 0,Y 484.802,Z 491.853,A -85,B 0,C 180,E1 -7045.548,E2 -7045.548} C_VEL
LIN {X 0,Y 484.333,Z 487.534,A -85,B 0,C 180,E1 -7046.289,E2 -7046.289} C_VEL
LIN {X 0,Y 481.708,Z 475.608,A -85,B 0,C 180,E1 -7048.454,E2 -7048.454} C_VEL
LIN {X 0,Y 481.648,Z 475.617,A -85,B 0,C 180,E1 -7051.688,E2 -7051.688} C_VEL
LIN {X 0,Y 481.694,Z 475.605,A -85,B 0,C 180,E1 -7054.682,E2 -7054.682} C_VEL
LIN {X 0,Y 481.658,Z 475.611,A -85,B 0,C 180,E1 -7058.007,E2 -7058.007} C_VEL
LIN {X 0,Y 481.659,Z 475.609,A -85,B 0,C 180,E1 -7061.042,E2 -7061.042} C_VEL
LIN {X 0,Y 481.657,Z 475.608,A -85,B 0,C 180,E1 -7064.458,E2 -7064.458} C_VEL
LIN {X 0,Y 481.65,Z 475.613,A -85,B 0,C 180,E1 -7067.839,E2 -7067.839} C_VEL
LIN {X 0,Y 481.658,Z 475.609,A -85,B 0,C 180,E1 -7069.018,E2 -7069.018} C_VEL
LIN {X 0,Y 480.998,Z 475.697,A -85,B 0,C 180,E1 -7069.716,E2 -7069.716} C_VEL
LIN {X 0,Y 478.154,Z 476.048,A -85,B 0,C 180,E1 -7070.849,E2 -7070.849} C_VEL
LIN {X 0,Y 475.735,Z 476.351,A -85,B 0,C 180,E1 -7071.762,E2 -7071.762} C_VEL
LIN {X 0,Y 474.68,Z 476.477,A -85,B 0,C 180,E1 -7072.467,E2 -7072.467} C_VEL
LIN {X 0,Y 474.586,Z 476.489,A -85,B 0,C 180,E1 -7072.706,E2 -7072.706} C_VEL
LIN {X 0,Y 474.639,Z 476.484,A -85,B 0,C 180,E1 -7076.016,E2 -7076.016} C_VEL
LIN {X 0,Y 474.606,Z 476.49,A -85,B 0,C 180,E1 -7079.19,E2 -7079.19} C_VEL
LIN {X 0,Y 474.648,Z 476.487,A -85,B 0,C 180,E1 -7081.717,E2 -7081.717} C_VEL
LIN {X 0,Y 474.671,Z 476.478,A -85,B 0,C 180,E1 -7084.578,E2 -7084.578} C_VEL
LIN {X 0,Y 474.603,Z 476.493,A -85,B 0,C 180,E1 -7087.355,E2 -7087.355} C_VEL
LIN {X 0,Y 474.659,Z 476.481,A -85,B 0,C 180,E1 -7090.09,E2 -7090.09} C_VEL
LIN {X 0,Y 474.653,Z 476.481,A -85,B 0,C 180,E1 -7092.774,E2 -7092.774} C_VEL
LIN {X 0,Y 474.655,Z 476.488,A -85,B 0,C 180,E1 -7095.421,E2 -7095.421} C_VEL
LIN {X 0,Y 474.706,Z 476.475,A -85,B 0,C 180,E1 -7098.038,E2 -7098.038} C_VEL
LIN {X 0,Y 474.731,Z 476.479,A -85,B 0,C 180,E1 -7101.486,E2 -7101.486} C_VEL
LIN {X 0,Y 474.781,Z 476.466,A -85,B 0,C 180,E1 -7104.052,E2 -7104.052} C_VEL
LIN {X 0,Y 474.897,Z 476.459,A -85,B 0,C 180,E1 -7107.455,E2 -7107.455} C_VEL
LIN {X 0,Y 474.914,Z 476.449,A -85,B 0,C 180,E1 -7110,E2 -7110} C_VEL
LIN {X 0,Y 474.897,Z 476.45,A -85,B 0,C 180,E1 -7112.545,E2 -7112.545} C_VEL
LIN {X 0,Y 474.773,Z 476.467,A -85,B 0,C 180,E1 -7115.948,E2 -7115.948} C_VEL
LIN {X 0,Y 474.73,Z 476.471,A -85,B 0,C 180,E1 -7118.513,E2 -7118.513} C_VEL
LIN {X 0,Y 474.706,Z 476.475,A -85,B 0,C 180,E1 -7121.962,E2 -7121.962} C_VEL
LIN {X 0,Y 474.702,Z 476.482,A -85,B 0,C 180,E1 -7125.456,E2 -7125.456} C_VEL
LIN {X 0,Y 474.667,Z 476.482,A -85,B 0,C 180,E1 -7129.01,E2 -7129.01} C_VEL
LIN {X 0,Y 474.593,Z 476.491,A -85,B 0,C 180,E1 -7131.729,E2 -7131.729} C_VEL
LIN {X 0,Y 474.661,Z 476.479,A -85,B 0,C 180,E1 -7134.493,E2 -7134.493} C_VEL
LIN {X 0,Y 474.701,Z 476.483,A -85,B 0,C 180,E1 -7137.339,E2 -7137.339} C_VEL
LIN {X 0,Y 474.606,Z 476.488,A -85,B 0,C 180,E1 -7140.81,E2 -7140.81} C_VEL
LIN {X 0,Y 474.639,Z 476.483,A -85,B 0,C 180,E1 -7143.984,E2 -7143.984} C_VEL
LIN {X 0,Y 474.574,Z 476.493,A -85,B 0,C 180,E1 -7146.899,E2 -7146.899} C_VEL
LIN {X 0,Y 474.629,Z 476.487,A -85,B 0,C 180,E1 -7149.648,E2 -7149.648} C_VEL
LIN {X 0,Y 474.637,Z 476.486,A -85,B 0,C 180,E1 -7152.932,E2 -7152.932} C_VEL
LIN {X 0,Y 474.611,Z 476.487,A -85,B 0,C 180,E1 -7155.895,E2 -7155.895} C_VEL
LIN {X 0,Y 474.629,Z 476.488,A -85,B 0,C 180,E1 -7159.041,E2 -7159.041} C_VEL
LIN {X 0,Y 474.612,Z 476.488,A -85,B 0,C 180,E1 -7161.704,E2 -7161.704} C_VEL
LIN {X 0,Y 474.627,Z 476.485,A -85,B 0,C 180,E1 -7164.726,E2 -7164.726} C_VEL
LIN {X 0,Y 474.638,Z 476.485,A -85,B 0,C 180,E1 -7167.788,E2 -7167.788} C_VEL
LIN {X 0,Y 474.627,Z 476.488,A -85,B 0,C 180,E1 -7170.885,E2 -7170.885} C_VEL
LIN {X 0,Y 474.731,Z 476.598,A -85,B 0,C 180,E1 -7172.771,E2 -7172.771} C_VEL
LIN {X 0,Y 477.498,Z 490.06,A -85,B 0,C 180,E1 -7174.966,E2 -7174.966} C_VEL
LIN {X 0,Y 477.37,Z 499.545,A -85,B 0,C 180,E1 -7176.397,E2 -7176.397} C_VEL
LIN {X 0,Y 476.745,Z 518.803,A -85,B 0,C 180,E1 -7179.28,E2 -7179.28} C_VEL
LIN {X 0,Y 476.103,Z 539.56,A -85,B 0,C 180,E1 -7182.386,E2 -7182.386} C_VEL
LIN {X 0,Y 475.888,Z 545.822,A -85,B 0,C 180,E1 -7183.319,E2 -7183.319} C_VEL
LIN {X 0,Y 478.01,Z 559.593,A -85,B 0,C 180,E1 -7183.639,E2 -7183.639} C_VEL
LIN {X 0,Y 477.126,Z 655.361,A -85,B 0,C 180,E1 -7185.226,E2 -7185.226} C_VEL
LIN {X 0,Y 476.833,Z 668.415,A -85,B 0,C 180,E1 -7185.598,E2 -7185.598} C_VEL
LIN {X 0,Y 476.447,Z 680.899,A -85,B 0,C 180,E1 -7186.131,E2 -7186.131} C_VEL
LIN {X 0,Y 476.098,Z 692.19,A -85,B 0,C 180,E1 -7186.774,E2 -7186.774} C_VEL
LIN {X 0,Y 475.793,Z 702.761,A -85,B 0,C 180,E1 -7187.536,E2 -7187.536} C_VEL
LIN {X 0,Y 475.344,Z 713.35,A -85,B 0,C 180,E1 -7188.487,E2 -7188.487} C_VEL
LIN {X 0,Y 474.922,Z 722.974,A -85,B 0,C 180,E1 -7189.556,E2 -7189.556} C_VEL
LIN {X 0,Y 474.568,Z 730.885,A -85,B 0,C 180,E1 -7190.625,E2 -7190.625} C_VEL
LIN {X 0,Y 474.249,Z 738.633,A -85,B 0,C 180,E1 -7191.907,E2 -7191.907} C_VEL
LIN {X 0,Y 474.024,Z 745.667,A -85,B 0,C 180,E1 -7193.395,E2 -7193.395} C_VEL
LIN {X 0,Y 473.965,Z 749.683,A -85,B 0,C 180,E1 -7194.469,E2 -7194.469} C_VEL
LIN {X 0,Y 473.834,Z 753.432,A -85,B 0,C 180,E1 -7195.747,E2 -7195.747} C_VEL
LIN {X 0,Y 473.837,Z 755.359,A -85,B 0,C 180,E1 -7196.599,E2 -7196.599} C_VEL
LIN {X 0,Y 473.762,Z 756.854,A -85,B 0,C 180,E1 -7197.449,E2 -7197.449} C_VEL
LIN {X 0,Y 473.727,Z 757.893,A -85,B 0,C 180,E1 -7198.3,E2 -7198.3} C_VEL
LIN {X 0,Y 473.669,Z 758.799,A -85,B 0,C 180,E1 -7200,E2 -7200} C_VEL
LIN {X 0,Y 473.689,Z 758.611,A -85,B 0,C 180,E1 -7200.85,E2 -7200.85} C_VEL
LIN {X 0,Y 473.727,Z 758.016,A -85,B 0,C 180,E1 -7201.7,E2 -7201.7} C_VEL
LIN {X 0,Y 473.762,Z 757.028,A -85,B 0,C 180,E1 -7202.551,E2 -7202.551} C_VEL
LIN {X 0,Y 473.836,Z 755.614,A -85,B 0,C 180,E1 -7203.401,E2 -7203.401} C_VEL
LIN {X 0,Y 473.806,Z 752.663,A -85,B 0,C 180,E1 -7204.68,E2 -7204.68} C_VEL
LIN {X 0,Y 474.004,Z 748.634,A -85,B 0,C 180,E1 -7205.957,E2 -7205.957} C_VEL
LIN {X 0,Y 474.124,Z 742.42,A -85,B 0,C 180,E1 -7207.452,E2 -7207.452} C_VEL
LIN {X 0,Y 474.419,Z 735.618,A -85,B 0,C 180,E1 -7208.734,E2 -7208.734} C_VEL
LIN {X 0,Y 474.748,Z 727.068,A -85,B 0,C 180,E1 -7210.017,E2 -7210.017} C_VEL
LIN {X 0,Y 475.066,Z 718.291,A -85,B 0,C 180,E1 -7211.088,E2 -7211.088} C_VEL
LIN {X 0,Y 475.516,Z 708.694,A -85,B 0,C 180,E1 -7212.046,E2 -7212.046} C_VEL
LIN {X 0,Y 475.894,Z 697.869,A -85,B 0,C 180,E1 -7212.918,E2 -7212.918} C_VEL
LIN {X 0,Y 476.257,Z 686.267,A -85,B 0,C 180,E1 -7213.657,E2 -7213.657} C_VEL
LIN {X 0,Y 476.627,Z 674.192,A -85,B 0,C 180,E1 -7214.245,E2 -7214.245} C_VEL
LIN {X 0,Y 476.96,Z 660.852,A -85,B 0,C 180,E1 -7214.698,E2 -7214.698} C_VEL
LIN {X 0,Y 477.164,Z 646.716,A -85,B 0,C 180,E1 -7214.991,E2 -7214.991} C_VEL
LIN {X 0,Y 478.115,Z 559.591,A -85,B 0,C 180,E1 -7216.47,E2 -7216.47} C_VEL
LIN {X 0,Y 476.019,Z 546.548,A -85,B 0,C 180,E1 -7216.795,E2 -7216.795} C_VEL
LIN {X 0,Y 476.606,Z 525.757,A -85,B 0,C 180,E1 -7219.826,E2 -7219.826} C_VEL
LIN {X 0,Y 477.185,Z 504.014,A -85,B 0,C 180,E1 -7222.973,E2 -7222.973} C_VEL
LIN {X 0,Y 477.49,Z 491.126,A -85,B 0,C 180,E1 -7224.802,E2 -7224.802} C_VEL
LIN {X 0,Y 476.26,Z 483.405,A -85,B 0,C 180,E1 -7225.982,E2 -7225.982} C_VEL
LIN {X 0,Y 474.706,Z 476.483,A -85,B 0,C 180,E1 -7227.081,E2 -7227.081} C_VEL
LIN {X 0,Y 474.608,Z 476.494,A -85,B 0,C 180,E1 -7230.23,E2 -7230.23} C_VEL
LIN {X 0,Y 474.645,Z 476.488,A -85,B 0,C 180,E1 -7233.22,E2 -7233.22} C_VEL
LIN {X 0,Y 474.591,Z 476.494,A -85,B 0,C 180,E1 -7236.323,E2 -7236.323} C_VEL
LIN {X 0,Y 474.63,Z 476.486,A -85,B 0,C 180,E1 -7239.648,E2 -7239.648} C_VEL
LIN {X 0,Y 474.617,Z 476.489,A -85,B 0,C 180,E1 -7242.934,E2 -7242.934} C_VEL
LIN {X 0,Y 474.617,Z 476.487,A -85,B 0,C 180,E1 -7245.896,E2 -7245.896} C_VEL
LIN {X 0,Y 474.634,Z 476.486,A -85,B 0,C 180,E1 -7249.04,E2 -7249.04} C_VEL
LIN {X 0,Y 474.612,Z 476.488,A -85,B 0,C 180,E1 -7251.704,E2 -7251.704} C_VEL
LIN {X 0,Y 474.632,Z 476.49,A -85,B 0,C 180,E1 -7254.726,E2 -7254.726} C_VEL
LIN {X 0,Y 474.64,Z 476.486,A -85,B 0,C 180,E1 -7257.788,E2 -7257.788} C_VEL
LIN {X 0,Y 474.634,Z 476.489,A -85,B 0,C 180,E1 -7260.883,E2 -7260.883} C_VEL
LIN {X 0,Y 474.73,Z 476.633,A -85,B 0,C 180,E1 -7262.75,E2 -7262.75} C_VEL
LIN {X 0,Y 478.29,Z 491.976,A -85,B 0,C 180,E1 -7265.236,E2 -7265.236} C_VEL
LIN {X 0,Y 478.635,Z 495.192,A -85,B 0,C 180,E1 -7265.724,E2 -7265.724} C_VEL
LIN {X 0,Y 477.353,Z 518.937,A -85,B 0,C 180,E1 -7269.082,E2 -7269.082} C_VEL
LIN {X 0,Y 477.081,Z 524.889,A -85,B 0,C 180,E1 -7269.908,E2 -7269.908} C_VEL
LIN {X 0,Y 479.731,Z 542.393,A -85,B 0,C 180,E1 -7270.309,E2 -7270.309} C_VEL
LIN {X 0,Y 478.316,Z 662.101,A -85,B 0,C 180,E1 -7272.249,E2 -7272.249} C_VEL
LIN {X 0,Y 477.918,Z 676.52,A -85,B 0,C 180,E1 -7272.648,E2 -7272.648} C_VEL
LIN {X 0,Y 477.578,Z 690.232,A -85,B 0,C 180,E1 -7273.204,E2 -7273.204} C_VEL
LIN {X 0,Y 477.094,Z 702.518,A -85,B 0,C 180,E1 -7273.856,E2 -7273.856} C_VEL
LIN {X 0,Y 476.46,Z 715.275,A -85,B 0,C 180,E1 -7274.712,E2 -7274.712} C_VEL
LIN {X 0,Y 475.9,Z 726.89,A -85,B 0,C 180,E1 -7275.679,E2 -7275.679} C_VEL
LIN {X 0,Y 475.368,Z 737.533,A -85,B 0,C 180,E1 -7276.753,E2 -7276.753} C_VEL
LIN {X 0,Y 474.954,Z 748.096,A -85,B 0,C 180,E1 -7278.044,E2 -7278.044} C_VEL
LIN {X 0,Y 474.541,Z 756.785,A -85,B 0,C 180,E1 -7279.331,E2 -7279.331} C_VEL
LIN {X 0,Y 474.204,Z 765.061,A -85,B 0,C 180,E1 -7280.832,E2 -7280.832} C_VEL
LIN {X 0,Y 473.954,Z 771.703,A -85,B 0,C 180,E1 -7282.331,E2 -7282.331} C_VEL
LIN {X 0,Y 473.872,Z 776.102,A -85,B 0,C 180,E1 -7283.555,E2 -7283.555} C_VEL
LIN {X 0,Y 473.825,Z 779.902,A -85,B 0,C 180,E1 -7284.894,E2 -7284.894} C_VEL
LIN {X 0,Y 473.786,Z 783.411,A -85,B 0,C 180,E1 -7286.598,E2 -7286.598} C_VEL
LIN {X 0,Y 473.721,Z 785.483,A -85,B 0,C 180,E1 -7288.3,E2 -7288.3} C_VEL
LIN {X 0,Y 473.668,Z 786.162,A -85,B 0,C 180,E1 -7290,E2 -7290} C_VEL
LIN {X 0,Y 473.721,Z 785.45,A -85,B 0,C 180,E1 -7291.7,E2 -7291.7} C_VEL
LIN {X 0,Y 473.786,Z 783.344,A -85,B 0,C 180,E1 -7293.402,E2 -7293.402} C_VEL
LIN {X 0,Y 473.825,Z 779.784,A -85,B 0,C 180,E1 -7295.106,E2 -7295.106} C_VEL
LIN {X 0,Y 473.892,Z 774.667,A -85,B 0,C 180,E1 -7296.814,E2 -7296.814} C_VEL
LIN {X 0,Y 474,Z 769.7,A -85,B 0,C 180,E1 -7298.098,E2 -7298.098} C_VEL
LIN {X 0,Y 474.268,Z 762.516,A -85,B 0,C 180,E1 -7299.597,E2 -7299.597} C_VEL
LIN {X 0,Y 474.677,Z 753.587,A -85,B 0,C 180,E1 -7301.097,E2 -7301.097} C_VEL
LIN {X 0,Y 475.051,Z 743.575,A -85,B 0,C 180,E1 -7302.468,E2 -7302.468} C_VEL
LIN {X 0,Y 475.519,Z 732.716,A -85,B 0,C 180,E1 -7303.679,E2 -7303.679} C_VEL
LIN {X 0,Y 476.049,Z 720.96,A -85,B 0,C 180,E1 -7304.754,E2 -7304.754} C_VEL
LIN {X 0,Y 476.697,Z 707.894,A -85,B 0,C 180,E1 -7305.718,E2 -7305.718} C_VEL
LIN {X 0,Y 477.188,Z 695.087,A -85,B 0,C 180,E1 -7306.468,E2 -7306.468} C_VEL
LIN {X 0,Y 477.638,Z 681.882,A -85,B 0,C 180,E1 -7307.064,E2 -7307.064} C_VEL
LIN {X 0,Y 478.032,Z 668.121,A -85,B 0,C 180,E1 -7307.514,E2 -7307.514} C_VEL
LIN {X 0,Y 478.293,Z 653.917,A -85,B 0,C 180,E1 -7307.807,E2 -7307.807} C_VEL
LIN {X 0,Y 479.502,Z 547.285,A -85,B 0,C 180,E1 -7309.554,E2 -7309.554} C_VEL
LIN {X 0,Y 479.375,Z 539.644,A -85,B 0,C 180,E1 -7309.696,E2 -7309.696} C_VEL
LIN {X 0,Y 477.126,Z 525.476,A -85,B 0,C 180,E1 -7310.055,E2 -7310.055} C_VEL
LIN {X 0,Y 478.516,Z 502.702,A -85,B 0,C 180,E1 -7313.363,E2 -7313.363} C_VEL
LIN {X 0,Y 479.03,Z 494.823,A -85,B 0,C 180,E1 -7314.547,E2 -7314.547} C_VEL
LIN {X 0,Y 476.605,Z 483.736,A -85,B 0,C 180,E1 -7316.492,E2 -7316.492} C_VEL
LIN {X 0,Y 474.677,Z 476.486,A -85,B 0,C 180,E1 -7317.89,E2 -7317.89} C_VEL
LIN {X 0,Y 474.602,Z 476.495,A -85,B 0,C 180,E1 -7321.218,E2 -7321.218} C_VEL
LIN {X 0,Y 474.634,Z 476.488,A -85,B 0,C 180,E1 -7324.241,E2 -7324.241} C_VEL
LIN {X 0,Y 474.592,Z 476.496,A -85,B 0,C 180,E1 -7327.384,E2 -7327.384} C_VEL
LIN {X 0,Y 474.63,Z 476.489,A -85,B 0,C 180,E1 -7329.648,E2 -7329.648} C_VEL
LIN {X 0,Y 474.638,Z 476.49,A -85,B 0,C 180,E1 -7332.932,E2 -7332.932} C_VEL
LIN {X 0,Y 474.612,Z 476.489,A -85,B 0,C 180,E1 -7335.895,E2 -7335.895} C_VEL
LIN {X 0,Y 474.63,Z 476.49,A -85,B 0,C 180,E1 -7339.041,E2 -7339.041} C_VEL
LIN {X 0,Y 474.613,Z 476.49,A -85,B 0,C 180,E1 -7341.704,E2 -7341.704} C_VEL
LIN {X 0,Y 474.629,Z 476.491,A -85,B 0,C 180,E1 -7344.726,E2 -7344.726} C_VEL
LIN {X 0,Y 474.64,Z 476.487,A -85,B 0,C 180,E1 -7347.788,E2 -7347.788} C_VEL
LIN {X 0,Y 474.628,Z 476.496,A -85,B 0,C 180,E1 -7350.885,E2 -7350.885} C_VEL
LIN {X 0,Y 474.726,Z 476.535,A -85,B 0,C 180,E1 -7352.835,E2 -7352.835} C_VEL
LIN {X 0,Y 477.423,Z 488.213,A -85,B 0,C 180,E1 -7355.194,E2 -7355.194} C_VEL
LIN {X 0,Y 478.358,Z 493.581,A -85,B 0,C 180,E1 -7356.208,E2 -7356.208} C_VEL
LIN {X 0,Y 477.308,Z 510.598,A -85,B 0,C 180,E1 -7359.08,E2 -7359.08} C_VEL
LIN {X 0,Y 476.401,Z 529.409,A -85,B 0,C 180,E1 -7362.175,E2 -7362.175} C_VEL
LIN {X 0,Y 475.905,Z 540.581,A -85,B 0,C 180,E1 -7363.982,E2 -7363.982} C_VEL
LIN {X 0,Y 478.609,Z 557.507,A -85,B 0,C 180,E1 -7364.424,E2 -7364.424} C_VEL
LIN {X 0,Y 477.215,Z 653.03,A -85,B 0,C 180,E1 -7366.154,E2 -7366.154} C_VEL
LIN {X 0,Y 476.894,Z 667.162,A -85,B 0,C 180,E1 -7366.593,E2 -7366.593} C_VEL
LIN {X 0,Y 476.605,Z 679.696,A -85,B 0,C 180,E1 -7367.163,E2 -7367.163} C_VEL
LIN {X 0,Y 476.208,Z 691.332,A -85,B 0,C 180,E1 -7367.86,E2 -7367.86} C_VEL
LIN {X 0,Y 475.708,Z 702.596,A -85,B 0,C 180,E1 -7368.711,E2 -7368.711} C_VEL
LIN {X 0,Y 475.238,Z 712.772,A -85,B 0,C 180,E1 -7369.67,E2 -7369.67} C_VEL
LIN {X 0,Y 474.877,Z 722.781,A -85,B 0,C 180,E1 -7370.846,E2 -7370.846} C_VEL
LIN {X 0,Y 474.44,Z 731.604,A -85,B 0,C 180,E1 -7372.124,E2 -7372.124} C_VEL
LIN {X 0,Y 474.292,Z 738.668,A -85,B 0,C 180,E1 -7373.416,E2 -7373.416} C_VEL
LIN {X 0,Y 474.02,Z 743.414,A -85,B 0,C 180,E1 -7374.47,E2 -7374.47} C_VEL
LIN {X 0,Y 473.982,Z 748,A -85,B 0,C 180,E1 -7375.748,E2 -7375.748} C_VEL
LIN {X 0,Y 473.879,Z 750.415,A -85,B 0,C 180,E1 -7376.599,E2 -7376.599} C_VEL
LIN {X 0,Y 473.816,Z 752.391,A -85,B 0,C 180,E1 -7377.45,E2 -7377.45} C_VEL
LIN {X 0,Y 473.765,Z 753.945,A -85,B 0,C 180,E1 -7378.3,E2 -7378.3} C_VEL
LIN {X 0,Y 473.69,Z 755.042,A -85,B 0,C 180,E1 -7379.15,E2 -7379.15} C_VEL
LIN {X 0,Y 473.688,Z 756.014,A -85,B 0,C 180,E1 -7380.85,E2 -7380.85} C_VEL
LIN {X 0,Y 473.727,Z 755.907,A -85,B 0,C 180,E1 -7381.7,E2 -7381.7} C_VEL
LIN {X 0,Y 473.759,Z 755.36,A -85,B 0,C 180,E1 -7382.551,E2 -7382.551} C_VEL
LIN {X 0,Y 473.817,Z 754.402,A -85,B 0,C 180,E1 -7383.401,E2 -7383.401} C_VEL
LIN {X 0,Y 473.773,Z 753.047,A -85,B 0,C 180,E1 -7384.254,E2 -7384.254} C_VEL
LIN {X 0,Y 473.91,Z 750.179,A -85,B 0,C 180,E1 -7385.532,E2 -7385.532} C_VEL
LIN {X 0,Y 473.922,Z 746.269,A -85,B 0,C 180,E1 -7386.813,E2 -7386.813} C_VEL
LIN {X 0,Y 474.1,Z 741.2,A -85,B 0,C 180,E1 -7388.096,E2 -7388.096} C_VEL
LIN {X 0,Y 474.324,Z 734.825,A -85,B 0,C 180,E1 -7389.38,E2 -7389.38} C_VEL
LIN {X 0,Y 474.625,Z 726.832,A -85,B 0,C 180,E1 -7390.667,E2 -7390.667} C_VEL
LIN {X 0,Y 475.062,Z 718.676,A -85,B 0,C 180,E1 -7391.737,E2 -7391.737} C_VEL
LIN {X 0,Y 475.33,Z 710.001,A -85,B 0,C 180,E1 -7392.686,E2 -7392.686} C_VEL
LIN {X 0,Y 475.819,Z 698.971,A -85,B 0,C 180,E1 -7393.67,E2 -7393.67} C_VEL
LIN {X 0,Y 476.269,Z 688.49,A -85,B 0,C 180,E1 -7394.419,E2 -7394.419} C_VEL
LIN {X 0,Y 476.685,Z 677.096,A -85,B 0,C 180,E1 -7395.061,E2 -7395.061} C_VEL
LIN {X 0,Y 476.934,Z 663.646,A -85,B 0,C 180,E1 -7395.628,E2 -7395.628} C_VEL
LIN {X 0,Y 477.29,Z 650.268,A -85,B 0,C 180,E1 -7396,E2 -7396} C_VEL
LIN {X 0,Y 478.352,Z 557.232,A -85,B 0,C 180,E1 -7397.565,E2 -7397.565} C_VEL
LIN {X 0,Y 475.79,Z 540.929,A -85,B 0,C 180,E1 -7397.964,E2 -7397.964} C_VEL
LIN {X 0,Y 476.407,Z 525.023,A -85,B 0,C 180,E1 -7400.509,E2 -7400.509} C_VEL
LIN {X 0,Y 477.17,Z 508.377,A -85,B 0,C 180,E1 -7403.203,E2 -7403.203} C_VEL
LIN {X 0,Y 477.95,Z 493.057,A -85,B 0,C 180,E1 -7405.708,E2 -7405.708} C_VEL
LIN {X 0,Y 477.12,Z 487.441,A -85,B 0,C 180,E1 -7406.697,E2 -7406.697} C_VEL
LIN {X 0,Y 474.667,Z 476.485,A -85,B 0,C 180,E1 -7408.734,E2 -7408.734} C_VEL
LIN {X 0,Y 474.639,Z 476.487,A -85,B 0,C 180,E1 -7412.212,E2 -7412.212} C_VEL
LIN {X 0,Y 474.63,Z 476.489,A -85,B 0,C 180,E1 -7415.274,E2 -7415.274} C_VEL
LIN {X 0,Y 474.614,Z 476.485,A -85,B 0,C 180,E1 -7418.457,E2 -7418.457} C_VEL
LIN {X 0,Y 474.63,Z 476.484,A -85,B 0,C 180,E1 -7420.959,E2 -7420.959} C_VEL
LIN {X 0,Y 474.608,Z 476.488,A -85,B 0,C 180,E1 -7424.105,E2 -7424.105} C_VEL
LIN {X 0,Y 474.617,Z 476.487,A -85,B 0,C 180,E1 -7427.066,E2 -7427.066} C_VEL
LIN {X 0,Y 474.62,Z 476.485,A -85,B 0,C 180,E1 -7430.354,E2 -7430.354} C_VEL
LIN {X 0,Y 474.586,Z 476.489,A -85,B 0,C 180,E1 -7432.706,E2 -7432.706} C_VEL
LIN {X 0,Y 473.905,Z 476.58,A -85,B 0,C 180,E1 -7433.415,E2 -7433.415} C_VEL
LIN {X 0,Y 471.078,Z 476.929,A -85,B 0,C 180,E1 -7434.567,E2 -7434.567} C_VEL
LIN {X 0,Y 468.693,Z 477.23,A -85,B 0,C 180,E1 -7435.495,E2 -7435.495} C_VEL
LIN {X 0,Y 467.663,Z 477.352,A -85,B 0,C 180,E1 -7436.212,E2 -7436.212} C_VEL
LIN {X 0,Y 467.574,Z 477.362,A -85,B 0,C 180,E1 -7436.455,E2 -7436.455} C_VEL
LIN {X 0,Y 467.571,Z 477.367,A -85,B 0,C 180,E1 -7439.266,E2 -7439.266} C_VEL
LIN {X 0,Y 467.635,Z 477.354,A -85,B 0,C 180,E1 -7442.461,E2 -7442.461} C_VEL
LIN {X 0,Y 467.604,Z 477.361,A -85,B 0,C 180,E1 -7445.113,E2 -7445.113} C_VEL
LIN {X 0,Y 467.536,Z 477.37,A -85,B 0,C 180,E1 -7447.926,E2 -7447.926} C_VEL
LIN {X 0,Y 467.626,Z 477.356,A -85,B 0,C 180,E1 -7450.692,E2 -7450.692} C_VEL
LIN {X 0,Y 467.652,Z 477.354,A -85,B 0,C 180,E1 -7454.114,E2 -7454.114} C_VEL
LIN {X 0,Y 467.656,Z 477.358,A -85,B 0,C 180,E1 -7457.642,E2 -7457.642} C_VEL
LIN {X 0,Y 467.668,Z 477.35,A -85,B 0,C 180,E1 -7460.485,E2 -7460.485} C_VEL
LIN {X 0,Y 467.714,Z 477.348,A -85,B 0,C 180,E1 -7463.096,E2 -7463.096} C_VEL
LIN {X 0,Y 467.727,Z 477.344,A -85,B 0,C 180,E1 -7464.827,E2 -7464.827} C_VEL
LIN {X 0,Y 467.862,Z 477.334,A -85,B 0,C 180,E1 -7467.417,E2 -7467.417} C_VEL
LIN {X 0,Y 467.885,Z 477.325,A -85,B 0,C 180,E1 -7470,E2 -7470} C_VEL
LIN {X 0,Y 467.862,Z 477.326,A -85,B 0,C 180,E1 -7472.583,E2 -7472.583} C_VEL
LIN {X 0,Y 467.737,Z 477.343,A -85,B 0,C 180,E1 -7476.037,E2 -7476.037} C_VEL
LIN {X 0,Y 467.683,Z 477.349,A -85,B 0,C 180,E1 -7478.643,E2 -7478.643} C_VEL
LIN {X 0,Y 467.658,Z 477.352,A -85,B 0,C 180,E1 -7482.145,E2 -7482.145} C_VEL
LIN {X 0,Y 467.641,Z 477.358,A -85,B 0,C 180,E1 -7485.695,E2 -7485.695} C_VEL
LIN {X 0,Y 467.619,Z 477.358,A -85,B 0,C 180,E1 -7488.765,E2 -7488.765} C_VEL
LIN {X 0,Y 467.583,Z 477.368,A -85,B 0,C 180,E1 -7491.269,E2 -7491.269} C_VEL
LIN {X 0,Y 467.575,Z 477.364,A -85,B 0,C 180,E1 -7493.943,E2 -7493.943} C_VEL
LIN {X 0,Y 467.618,Z 477.358,A -85,B 0,C 180,E1 -7496.8,E2 -7496.8} C_VEL
LIN {X 0,Y 467.556,Z 477.368,A -85,B 0,C 180,E1 -7499.738,E2 -7499.738} C_VEL
LIN {X 0,Y 467.585,Z 477.362,A -85,B 0,C 180,E1 -7502.758,E2 -7502.758} C_VEL
LIN {X 0,Y 467.555,Z 477.366,A -85,B 0,C 180,E1 -7505.89,E2 -7505.89} C_VEL
LIN {X 0,Y 467.584,Z 477.367,A -85,B 0,C 180,E1 -7509.145,E2 -7509.145} C_VEL
LIN {X 0,Y 467.588,Z 477.361,A -85,B 0,C 180,E1 -7512.567,E2 -7512.567} C_VEL
LIN {X 0,Y 467.572,Z 477.367,A -85,B 0,C 180,E1 -7515.053,E2 -7515.053} C_VEL
LIN {X 0,Y 467.59,Z 477.367,A -85,B 0,C 180,E1 -7517.44,E2 -7517.44} C_VEL
LIN {X 0,Y 467.584,Z 477.364,A -85,B 0,C 180,E1 -7520.855,E2 -7520.855} C_VEL
LIN {X 0,Y 467.562,Z 477.363,A -85,B 0,C 180,E1 -7524.261,E2 -7524.261} C_VEL
LIN {X 0,Y 467.584,Z 477.369,A -85,B 0,C 180,E1 -7527.321,E2 -7527.321} C_VEL
LIN {X 0,Y 467.573,Z 477.365,A -85,B 0,C 180,E1 -7530.667,E2 -7530.667} C_VEL
LIN {X 0,Y 467.666,Z 477.517,A -85,B 0,C 180,E1 -7532.551,E2 -7532.551} C_VEL
LIN {X 0,Y 470.561,Z 491.216,A -85,B 0,C 180,E1 -7534.808,E2 -7534.808} C_VEL
LIN {X 0,Y 470.651,Z 496.57,A -85,B 0,C 180,E1 -7535.628,E2 -7535.628} C_VEL
LIN {X 0,Y 469.961,Z 515.624,A -85,B 0,C 180,E1 -7538.507,E2 -7538.507} C_VEL
LIN {X 0,Y 469.316,Z 535.121,A -85,B 0,C 180,E1 -7541.445,E2 -7541.445} C_VEL
LIN {X 0,Y 468.959,Z 546.009,A -85,B 0,C 180,E1 -7543.081,E2 -7543.081} C_VEL
LIN {X 0,Y 471.225,Z 561.125,A -85,B 0,C 180,E1 -7543.431,E2 -7543.431} C_VEL
LIN {X 0,Y 470.231,Z 655.42,A -85,B 0,C 180,E1 -7545.032,E2 -7545.032} C_VEL
LIN {X 0,Y 469.92,Z 667.671,A -85,B 0,C 180,E1 -7545.382,E2 -7545.382} C_VEL
LIN {X 0,Y 469.552,Z 680.455,A -85,B 0,C 180,E1 -7545.923,E2 -7545.923} C_VEL
LIN {X 0,Y 469.101,Z 693.548,A -85,B 0,C 180,E1 -7546.683,E2 -7546.683} C_VEL
LIN {X 0,Y 468.737,Z 704.201,A -85,B 0,C 180,E1 -7547.483,E2 -7547.483} C_VEL
LIN {X 0,Y 468.248,Z 715.307,A -85,B 0,C 180,E1 -7548.529,E2 -7548.529} C_VEL
LIN {X 0,Y 467.842,Z 724.658,A -85,B 0,C 180,E1 -7549.615,E2 -7549.615} C_VEL
LIN {X 0,Y 467.438,Z 733.656,A -85,B 0,C 180,E1 -7550.917,E2 -7550.917} C_VEL
LIN {X 0,Y 467.113,Z 740.896,A -85,B 0,C 180,E1 -7552.218,E2 -7552.218} C_VEL
LIN {X 0,Y 466.946,Z 747.209,A -85,B 0,C 180,E1 -7553.658,E2 -7553.658} C_VEL
LIN {X 0,Y 466.797,Z 751.208,A -85,B 0,C 180,E1 -7554.817,E2 -7554.817} C_VEL
LIN {X 0,Y 466.737,Z 753.578,A -85,B 0,C 180,E1 -7555.682,E2 -7555.682} C_VEL
LIN {X 0,Y 466.767,Z 755.516,A -85,B 0,C 180,E1 -7556.547,E2 -7556.547} C_VEL
LIN {X 0,Y 466.683,Z 757.026,A -85,B 0,C 180,E1 -7557.411,E2 -7557.411} C_VEL
LIN {X 0,Y 466.62,Z 758.728,A -85,B 0,C 180,E1 -7559.137,E2 -7559.137} C_VEL
LIN {X 0,Y 466.598,Z 758.991,A -85,B 0,C 180,E1 -7560,E2 -7560} C_VEL
LIN {X 0,Y 466.62,Z 758.807,A -85,B 0,C 180,E1 -7560.863,E2 -7560.863} C_VEL
LIN {X 0,Y 466.683,Z 757.225,A -85,B 0,C 180,E1 -7562.589,E2 -7562.589} C_VEL
LIN {X 0,Y 466.767,Z 755.807,A -85,B 0,C 180,E1 -7563.453,E2 -7563.453} C_VEL
LIN {X 0,Y 466.728,Z 752.845,A -85,B 0,C 180,E1 -7564.751,E2 -7564.751} C_VEL
LIN {X 0,Y 466.929,Z 748.801,A -85,B 0,C 180,E1 -7566.048,E2 -7566.048} C_VEL
LIN {X 0,Y 467.077,Z 742.559,A -85,B 0,C 180,E1 -7567.566,E2 -7567.566} C_VEL
LIN {X 0,Y 467.373,Z 735.727,A -85,B 0,C 180,E1 -7568.866,E2 -7568.866} C_VEL
LIN {X 0,Y 467.753,Z 727.13,A -85,B 0,C 180,E1 -7570.169,E2 -7570.169} C_VEL
LIN {X 0,Y 468.1,Z 718.308,A -85,B 0,C 180,E1 -7571.255,E2 -7571.255} C_VEL
LIN {X 0,Y 468.614,Z 707.673,A -85,B 0,C 180,E1 -7572.315,E2 -7572.315} C_VEL
LIN {X 0,Y 469.01,Z 696.756,A -85,B 0,C 180,E1 -7573.188,E2 -7573.188} C_VEL
LIN {X 0,Y 469.331,Z 686.195,A -85,B 0,C 180,E1 -7573.862,E2 -7573.862} C_VEL
LIN {X 0,Y 469.754,Z 674.065,A -85,B 0,C 180,E1 -7574.458,E2 -7574.458} C_VEL
LIN {X 0,Y 470.097,Z 660.682,A -85,B 0,C 180,E1 -7574.917,E2 -7574.917} C_VEL
LIN {X 0,Y 470.307,Z 646.457,A -85,B 0,C 180,E1 -7575.215,E2 -7575.215} C_VEL
LIN {X 0,Y 471.281,Z 559.782,A -85,B 0,C 180,E1 -7576.731,E2 -7576.731} C_VEL
LIN {X 0,Y 469.169,Z 546.733,A -85,B 0,C 180,E1 -7577.079,E2 -7577.079} C_VEL
LIN {X 0,Y 469.833,Z 524.454,A -85,B 0,C 180,E1 -7580.352,E2 -7580.352} C_VEL
LIN {X 0,Y 470.355,Z 505.655,A -85,B 0,C 180,E1 -7583.093,E2 -7583.093} C_VEL
LIN {X 0,Y 470.696,Z 492.764,A -85,B 0,C 180,E1 -7584.949,E2 -7584.949} C_VEL
LIN {X 0,Y 469.204,Z 483.973,A -85,B 0,C 180,E1 -7586.308,E2 -7586.308} C_VEL
LIN {X 0,Y 467.657,Z 477.36,A -85,B 0,C 180,E1 -7587.399,E2 -7587.399} C_VEL
LIN {X 0,Y 467.571,Z 477.371,A -85,B 0,C 180,E1 -7591.045,E2 -7591.045} C_VEL
LIN {X 0,Y 467.591,Z 477.368,A -85,B 0,C 180,E1 -7594.242,E2 -7594.242} C_VEL
LIN {X 0,Y 467.55,Z 477.37,A -85,B 0,C 180,E1 -7597.186,E2 -7597.186} C_VEL
LIN {X 0,Y 467.579,Z 477.367,A -85,B 0,C 180,E1 -7600.264,E2 -7600.264} C_VEL
LIN {X 0,Y 467.588,Z 477.367,A -85,B 0,C 180,E1 -7602.567,E2 -7602.567} C_VEL
LIN {X 0,Y 467.573,Z 477.365,A -85,B 0,C 180,E1 -7605.053,E2 -7605.053} C_VEL
LIN {X 0,Y 467.591,Z 477.362,A -85,B 0,C 180,E1 -7607.44,E2 -7607.44} C_VEL
LIN {X 0,Y 467.584,Z 477.365,A -85,B 0,C 180,E1 -7610.855,E2 -7610.855} C_VEL
LIN {X 0,Y 467.565,Z 477.369,A -85,B 0,C 180,E1 -7614.26,E2 -7614.26} C_VEL
LIN {X 0,Y 467.585,Z 477.364,A -85,B 0,C 180,E1 -7617.321,E2 -7617.321} C_VEL
LIN {X 0,Y 467.58,Z 477.368,A -85,B 0,C 180,E1 -7620.666,E2 -7620.666} C_VEL
LIN {X 0,Y 467.666,Z 477.493,A -85,B 0,C 180,E1 -7622.454,E2 -7622.454} C_VEL
LIN {X 0,Y 471.065,Z 491.94,A -85,B 0,C 180,E1 -7624.837,E2 -7624.837} C_VEL
LIN {X 0,Y 471.826,Z 496.266,A -85,B 0,C 180,E1 -7625.519,E2 -7625.519} C_VEL
LIN {X 0,Y 470.447,Z 520.441,A -85,B 0,C 180,E1 -7628.99,E2 -7628.99} C_VEL
LIN {X 0,Y 470.197,Z 524.902,A -85,B 0,C 180,E1 -7629.623,E2 -7629.623} C_VEL
LIN {X 0,Y 472.965,Z 542.105,A -85,B 0,C 180,E1 -7630.038,E2 -7630.038} C_VEL
LIN {X 0,Y 471.446,Z 662.597,A -85,B 0,C 180,E1 -7632.037,E2 -7632.037} C_VEL
LIN {X 0,Y 471.058,Z 676.804,A -85,B 0,C 180,E1 -7632.443,E2 -7632.443} C_VEL
LIN {X 0,Y 470.668,Z 690.905,A -85,B 0,C 180,E1 -7633.031,E2 -7633.031} C_VEL
LIN {X 0,Y 470.145,Z 703.503,A -85,B 0,C 180,E1 -7633.723,E2 -7633.723} C_VEL
LIN {X 0,Y 469.479,Z 716.048,A -85,B 0,C 180,E1 -7634.591,E2 -7634.591} C_VEL
LIN {X 0,Y 468.895,Z 727.513,A -85,B 0,C 180,E1 -7635.571,E2 -7635.571} C_VEL
LIN {X 0,Y 468.295,Z 739.008,A -85,B 0,C 180,E1 -7636.77,E2 -7636.77} C_VEL
LIN {X 0,Y 467.848,Z 749.237,A -85,B 0,C 180,E1 -7638.08,E2 -7638.08} C_VEL
LIN {X 0,Y 467.441,Z 757.704,A -85,B 0,C 180,E1 -7639.387,E2 -7639.387} C_VEL
LIN {X 0,Y 467.115,Z 765.774,A -85,B 0,C 180,E1 -7640.91,E2 -7640.91} C_VEL
LIN {X 0,Y 466.869,Z 771.422,A -85,B 0,C 180,E1 -7642.214,E2 -7642.214} C_VEL
LIN {X 0,Y 466.799,Z 776.156,A -85,B 0,C 180,E1 -7643.554,E2 -7643.554} C_VEL
LIN {X 0,Y 466.734,Z 779.653,A -85,B 0,C 180,E1 -7644.816,E2 -7644.816} C_VEL
LIN {X 0,Y 466.68,Z 783.176,A -85,B 0,C 180,E1 -7646.547,E2 -7646.547} C_VEL
LIN {X 0,Y 466.628,Z 785.256,A -85,B 0,C 180,E1 -7648.274,E2 -7648.274} C_VEL
LIN {X 0,Y 466.597,Z 785.939,A -85,B 0,C 180,E1 -7650,E2 -7650} C_VEL
LIN {X 0,Y 466.628,Z 785.218,A -85,B 0,C 180,E1 -7651.726,E2 -7651.726} C_VEL
LIN {X 0,Y 466.68,Z 783.093,A -85,B 0,C 180,E1 -7653.454,E2 -7653.454} C_VEL
LIN {X 0,Y 466.734,Z 779.515,A -85,B 0,C 180,E1 -7655.184,E2 -7655.184} C_VEL
LIN {X 0,Y 466.822,Z 774.374,A -85,B 0,C 180,E1 -7656.918,E2 -7656.918} C_VEL
LIN {X 0,Y 466.936,Z 769.378,A -85,B 0,C 180,E1 -7658.221,E2 -7658.221} C_VEL
LIN {X 0,Y 467.204,Z 762.15,A -85,B 0,C 180,E1 -7659.743,E2 -7659.743} C_VEL
LIN {X 0,Y 467.633,Z 753.179,A -85,B 0,C 180,E1 -7661.267,E2 -7661.267} C_VEL
LIN {X 0,Y 468.096,Z 742.821,A -85,B 0,C 180,E1 -7662.692,E2 -7662.692} C_VEL
LIN {X 0,Y 468.556,Z 732.195,A -85,B 0,C 180,E1 -7663.886,E2 -7663.886} C_VEL
LIN {X 0,Y 469.096,Z 720.357,A -85,B 0,C 180,E1 -7664.978,E2 -7664.978} C_VEL
LIN {X 0,Y 469.724,Z 708.82,A -85,B 0,C 180,E1 -7665.846,E2 -7665.846} C_VEL
LIN {X 0,Y 470.255,Z 695.992,A -85,B 0,C 180,E1 -7666.625,E2 -7666.625} C_VEL
LIN {X 0,Y 470.748,Z 682.713,A -85,B 0,C 180,E1 -7667.246,E2 -7667.246} C_VEL
LIN {X 0,Y 471.135,Z 669.671,A -85,B 0,C 180,E1 -7667.694,E2 -7667.694} C_VEL
LIN {X 0,Y 471.463,Z 655.217,A -85,B 0,C 180,E1 -7668.018,E2 -7668.018} C_VEL
LIN {X 0,Y 472.695,Z 554.698,A -85,B 0,C 180,E1 -7669.709,E2 -7669.709} C_VEL
LIN {X 0,Y 472.724,Z 540.789,A -85,B 0,C 180,E1 -7669.962,E2 -7669.962} C_VEL
LIN {X 0,Y 470.33,Z 525.733,A -85,B 0,C 180,E1 -7670.358,E2 -7670.358} C_VEL
LIN {X 0,Y 471.837,Z 503.123,A -85,B 0,C 180,E1 -7673.714,E2 -7673.714} C_VEL
LIN {X 0,Y 472.206,Z 496.215,A -85,B 0,C 180,E1 -7674.785,E2 -7674.785} C_VEL
LIN {X 0,Y 469.932,Z 485.874,A -85,B 0,C 180,E1 -7676.658,E2 -7676.658} C_VEL
LIN {X 0,Y 467.598,Z 477.369,A -85,B 0,C 180,E1 -7678.35,E2 -7678.35} C_VEL
LIN {X 0,Y 467.586,Z 477.369,A -85,B 0,C 180,E1 -7681.74,E2 -7681.74} C_VEL
LIN {X 0,Y 467.566,Z 477.37,A -85,B 0,C 180,E1 -7684.833,E2 -7684.833} C_VEL
LIN {X 0,Y 467.567,Z 477.368,A -85,B 0,C 180,E1 -7688.045,E2 -7688.045} C_VEL
LIN {X 0,Y 467.584,Z 477.368,A -85,B 0,C 180,E1 -7691.278,E2 -7691.278} C_VEL
LIN {X 0,Y 467.57,Z 477.367,A -85,B 0,C 180,E1 -7693.823,E2 -7693.823} C_VEL
LIN {X 0,Y 467.559,Z 477.368,A -85,B 0,C 180,E1 -7696.256,E2 -7696.256} C_VEL
LIN {X 0,Y 467.581,Z 477.369,A -85,B 0,C 180,E1 -7698.723,E2 -7698.723} C_VEL
LIN {X 0,Y 467.568,Z 477.367,A -85,B 0,C 180,E1 -7701.956,E2 -7701.956} C_VEL
LIN {X 0,Y 467.569,Z 477.37,A -85,B 0,C 180,E1 -7705.168,E2 -7705.168} C_VEL
LIN {X 0,Y 467.587,Z 477.367,A -85,B 0,C 180,E1 -7708.26,E2 -7708.26} C_VEL
LIN {X 0,Y 467.581,Z 477.374,A -85,B 0,C 180,E1 -7711.251,E2 -7711.251} C_VEL
LIN {X 0,Y 467.649,Z 477.428,A -85,B 0,C 180,E1 -7712.389,E2 -7712.389} C_VEL
LIN {X 0,Y 470.171,Z 487.666,A -85,B 0,C 180,E1 -7714.548,E2 -7714.548} C_VEL
LIN {X 0,Y 471.565,Z 495.011,A -85,B 0,C 180,E1 -7715.996,E2 -7715.996} C_VEL
LIN {X 0,Y 470.678,Z 508.42,A -85,B 0,C 180,E1 -7718.312,E2 -7718.312} C_VEL
LIN {X 0,Y 469.631,Z 528.435,A -85,B 0,C 180,E1 -7721.684,E2 -7721.684} C_VEL
LIN {X 0,Y 469.059,Z 540.703,A -85,B 0,C 180,E1 -7723.666,E2 -7723.666} C_VEL
LIN {X 0,Y 471.869,Z 557.343,A -85,B 0,C 180,E1 -7724.133,E2 -7724.133} C_VEL
LIN {X 0,Y 470.632,Z 640.882,A -85,B 0,C 180,E1 -7725.68,E2 -7725.68} C_VEL
LIN {X 0,Y 470.297,Z 656.185,A -85,B 0,C 180,E1 -7726.001,E2 -7726.001} C_VEL
LIN {X 0,Y 469.998,Z 668.993,A -85,B 0,C 180,E1 -7726.441,E2 -7726.441} C_VEL
LIN {X 0,Y 469.675,Z 681.206,A -85,B 0,C 180,E1 -7727.029,E2 -7727.029} C_VEL
LIN {X 0,Y 469.246,Z 693.262,A -85,B 0,C 180,E1 -7727.787,E2 -7727.787} C_VEL
LIN {X 0,Y 468.686,Z 704.117,A -85,B 0,C 180,E1 -7728.649,E2 -7728.649} C_VEL
LIN {X 0,Y 468.213,Z 713.996,A -85,B 0,C 180,E1 -7729.623,E2 -7729.623} C_VEL
LIN {X 0,Y 467.872,Z 723.025,A -85,B 0,C 180,E1 -7730.707,E2 -7730.707} C_VEL
LIN {X 0,Y 467.414,Z 731.854,A -85,B 0,C 180,E1 -7732.005,E2 -7732.005} C_VEL
LIN {X 0,Y 467.244,Z 739.259,A -85,B 0,C 180,E1 -7733.387,E2 -7733.387} C_VEL
LIN {X 0,Y 466.849,Z 745.318,A -85,B 0,C 180,E1 -7734.818,E2 -7734.818} C_VEL
LIN {X 0,Y 466.867,Z 749.524,A -85,B 0,C 180,E1 -7736.116,E2 -7736.116} C_VEL
LIN {X 0,Y 466.733,Z 752.653,A -85,B 0,C 180,E1 -7737.411,E2 -7737.411} C_VEL
LIN {X 0,Y 466.671,Z 754.204,A -85,B 0,C 180,E1 -7738.274,E2 -7738.274} C_VEL
LIN {X 0,Y 466.621,Z 755.29,A -85,B 0,C 180,E1 -7739.137,E2 -7739.137} C_VEL
LIN {X 0,Y 466.619,Z 756.245,A -85,B 0,C 180,E1 -7740.863,E2 -7740.863} C_VEL
LIN {X 0,Y 466.634,Z 756.125,A -85,B 0,C 180,E1 -7741.726,E2 -7741.726} C_VEL
LIN {X 0,Y 466.679,Z 755.559,A -85,B 0,C 180,E1 -7742.589,E2 -7742.589} C_VEL
LIN {X 0,Y 466.728,Z 754.588,A -85,B 0,C 180,E1 -7743.453,E2 -7743.453} C_VEL
LIN {X 0,Y 466.682,Z 753.216,A -85,B 0,C 180,E1 -7744.318,E2 -7744.318} C_VEL
LIN {X 0,Y 466.823,Z 750.316,A -85,B 0,C 180,E1 -7745.616,E2 -7745.616} C_VEL
LIN {X 0,Y 466.849,Z 746.366,A -85,B 0,C 180,E1 -7746.917,E2 -7746.917} C_VEL
LIN {X 0,Y 467.074,Z 740.275,A -85,B 0,C 180,E1 -7748.436,E2 -7748.436} C_VEL
LIN {X 0,Y 467.348,Z 733.566,A -85,B 0,C 180,E1 -7749.74,E2 -7749.74} C_VEL
LIN {X 0,Y 467.738,Z 725.229,A -85,B 0,C 180,E1 -7751.045,E2 -7751.045} C_VEL
LIN {X 0,Y 468.11,Z 716.699,A -85,B 0,C 180,E1 -7752.133,E2 -7752.133} C_VEL
LIN {X 0,Y 468.526,Z 706.18,A -85,B 0,C 180,E1 -7753.224,E2 -7753.224} C_VEL
LIN {X 0,Y 469.094,Z 694.347,A -85,B 0,C 180,E1 -7754.201,E2 -7754.201} C_VEL
LIN {X 0,Y 469.536,Z 682.6,A -85,B 0,C 180,E1 -7754.963,E2 -7754.963} C_VEL
LIN {X 0,Y 469.937,Z 669.218,A -85,B 0,C 180,E1 -7755.616,E2 -7755.616} C_VEL
LIN {X 0,Y 470.247,Z 656.685,A -85,B 0,C 180,E1 -7756.051,E2 -7756.051} C_VEL
LIN {X 0,Y 470.512,Z 640.953,A -85,B 0,C 180,E1 -7756.376,E2 -7756.376} C_VEL
LIN {X 0,Y 471.506,Z 557.536,A -85,B 0,C 180,E1 -7757.809,E2 -7757.809} C_VEL
LIN {X 0,Y 468.885,Z 540.809,A -85,B 0,C 180,E1 -7758.238,E2 -7758.238} C_VEL
LIN {X 0,Y 469.602,Z 523.488,A -85,B 0,C 180,E1 -7761.05,E2 -7761.05} C_VEL
LIN {X 0,Y 470.531,Z 505.057,A -85,B 0,C 180,E1 -7764.076,E2 -7764.076} C_VEL
LIN {X 0,Y 471.027,Z 493.342,A -85,B 0,C 180,E1 -7766.03,E2 -7766.03} C_VEL
LIN {X 0,Y 468.215,Z 480.082,A -85,B 0,C 180,E1 -7768.465,E2 -7768.465} C_VEL
LIN {X 0,Y 467.617,Z 477.364,A -85,B 0,C 180,E1 -7768.986,E2 -7768.986} C_VEL
LIN {X 0,Y 467.586,Z 477.368,A -85,B 0,C 180,E1 -7771.74,E2 -7771.74} C_VEL
LIN {X 0,Y 467.569,Z 477.366,A -85,B 0,C 180,E1 -7774.832,E2 -7774.832} C_VEL
LIN {X 0,Y 467.568,Z 477.366,A -85,B 0,C 180,E1 -7778.044,E2 -7778.044} C_VEL
LIN {X 0,Y 467.58,Z 477.365,A -85,B 0,C 180,E1 -7781.277,E2 -7781.277} C_VEL
LIN {X 0,Y 467.554,Z 477.37,A -85,B 0,C 180,E1 -7783.82,E2 -7783.82} C_VEL
LIN {X 0,Y 467.556,Z 477.365,A -85,B 0,C 180,E1 -7786.255,E2 -7786.255} C_VEL
LIN {X 0,Y 467.58,Z 477.361,A -85,B 0,C 180,E1 -7788.723,E2 -7788.723} C_VEL
LIN {X 0,Y 467.567,Z 477.366,A -85,B 0,C 180,E1 -7791.955,E2 -7791.955} C_VEL
LIN {X 0,Y 467.566,Z 477.366,A -85,B 0,C 180,E1 -7795.167,E2 -7795.167} C_VEL
LIN {X 0,Y 467.574,Z 477.362,A -85,B 0,C 180,E1 -7796.455,E2 -7796.455} C_VEL
LIN {X 0,Y 466.886,Z 477.453,A -85,B 0,C 180,E1 -7797.174,E2 -7797.174} C_VEL
LIN {X 0,Y 464.008,Z 477.809,A -85,B 0,C 180,E1 -7798.341,E2 -7798.341} C_VEL
LIN {X 0,Y 461.6,Z 478.111,A -85,B 0,C 180,E1 -7799.283,E2 -7799.283} C_VEL
LIN {X 0,Y 460.591,Z 478.235,A -85,B 0,C 180,E1 -7800.011,E2 -7800.011} C_VEL
LIN {X 0,Y 460.521,Z 478.241,A -85,B 0,C 180,E1 -7800.257,E2 -7800.257} C_VEL
LIN {X 0,Y 460.575,Z 478.234,A -85,B 0,C 180,E1 -7802.756,E2 -7802.756} C_VEL
LIN {X 0,Y 460.543,Z 478.244,A -85,B 0,C 180,E1 -7805.668,E2 -7805.668} C_VEL
LIN {X 0,Y 460.523,Z 478.24,A -85,B 0,C 180,E1 -7808.578,E2 -7808.578} C_VEL
LIN {X 0,Y 460.593,Z 478.237,A -85,B 0,C 180,E1 -7811.311,E2 -7811.311} C_VEL
LIN {X 0,Y 460.606,Z 478.232,A -85,B 0,C 180,E1 -7814.059,E2 -7814.059} C_VEL
LIN {X 0,Y 460.611,Z 478.235,A -85,B 0,C 180,E1 -7817.666,E2 -7817.666} C_VEL
LIN {X 0,Y 460.631,Z 478.232,A -85,B 0,C 180,E1 -7821.224,E2 -7821.224} C_VEL
LIN {X 0,Y 460.712,Z 478.22,A -85,B 0,C 180,E1 -7823.87,E2 -7823.87} C_VEL
LIN {X 0,Y 460.827,Z 478.21,A -85,B 0,C 180,E1 -7827.378,E2 -7827.378} C_VEL
LIN {X 0,Y 460.855,Z 478.201,A -85,B 0,C 180,E1 -7830,E2 -7830} C_VEL
LIN {X 0,Y 460.827,Z 478.203,A -85,B 0,C 180,E1 -7832.622,E2 -7832.622} C_VEL
LIN {X 0,Y 460.703,Z 478.219,A -85,B 0,C 180,E1 -7836.13,E2 -7836.13} C_VEL
LIN {X 0,Y 460.63,Z 478.228,A -85,B 0,C 180,E1 -7838.776,E2 -7838.776} C_VEL
LIN {X 0,Y 460.615,Z 478.229,A -85,B 0,C 180,E1 -7842.445,E2 -7842.445} C_VEL
LIN {X 0,Y 460.602,Z 478.232,A -85,B 0,C 180,E1 -7845.998,E2 -7845.998} C_VEL
LIN {X 0,Y 460.573,Z 478.236,A -85,B 0,C 180,E1 -7848.902,E2 -7848.902} C_VEL
LIN {X 0,Y 460.518,Z 478.248,A -85,B 0,C 180,E1 -7851.486,E2 -7851.486} C_VEL
LIN {X 0,Y 460.544,Z 478.238,A -85,B 0,C 180,E1 -7854.332,E2 -7854.332} C_VEL
LIN {X 0,Y 460.581,Z 478.24,A -85,B 0,C 180,E1 -7857.243,E2 -7857.243} C_VEL
LIN {X 0,Y 460.512,Z 478.242,A -85,B 0,C 180,E1 -7860.24,E2 -7860.24} C_VEL
LIN {X 0,Y 460.53,Z 478.248,A -85,B 0,C 180,E1 -7863.325,E2 -7863.325} C_VEL
LIN {X 0,Y 460.478,Z 478.246,A -85,B 0,C 180,E1 -7866.529,E2 -7866.529} C_VEL
LIN {X 0,Y 460.56,Z 478.238,A -85,B 0,C 180,E1 -7869.86,E2 -7869.86} C_VEL
LIN {X 0,Y 460.519,Z 478.244,A -85,B 0,C 180,E1 -7872.901,E2 -7872.901} C_VEL
LIN {X 0,Y 460.513,Z 478.244,A -85,B 0,C 180,E1 -7875.83,E2 -7875.83} C_VEL
LIN {X 0,Y 460.533,Z 478.243,A -85,B 0,C 180,E1 -7878.989,E2 -7878.989} C_VEL
LIN {X 0,Y 460.529,Z 478.248,A -85,B 0,C 180,E1 -7881.267,E2 -7881.267} C_VEL
LIN {X 0,Y 460.513,Z 478.242,A -85,B 0,C 180,E1 -7884.555,E2 -7884.555} C_VEL
LIN {X 0,Y 460.534,Z 478.243,A -85,B 0,C 180,E1 -7887.716,E2 -7887.716} C_VEL
LIN {X 0,Y 460.542,Z 478.241,A -85,B 0,C 180,E1 -7890.769,E2 -7890.769} C_VEL
LIN {X 0,Y 460.605,Z 478.272,A -85,B 0,C 180,E1 -7892.302,E2 -7892.302} C_VEL
LIN {X 0,Y 463.585,Z 492.362,A -85,B 0,C 180,E1 -7894.642,E2 -7894.642} C_VEL
LIN {X 0,Y 463.773,Z 497.215,A -85,B 0,C 180,E1 -7895.401,E2 -7895.401} C_VEL
LIN {X 0,Y 463.038,Z 517.053,A -85,B 0,C 180,E1 -7898.419,E2 -7898.419} C_VEL
LIN {X 0,Y 462.361,Z 536.566,A -85,B 0,C 180,E1 -7901.385,E2 -7901.385} C_VEL
LIN {X 0,Y 462.054,Z 546.115,A -85,B 0,C 180,E1 -7902.831,E2 -7902.831} C_VEL
LIN {X 0,Y 464.376,Z 561.997,A -85,B 0,C 180,E1 -7903.21,E2 -7903.21} C_VEL
LIN {X 0,Y 463.333,Z 656.663,A -85,B 0,C 180,E1 -7904.86,E2 -7904.86} C_VEL
LIN {X 0,Y 462.979,Z 669.973,A -85,B 0,C 180,E1 -7905.27,E2 -7905.27} C_VEL
LIN {X 0,Y 462.556,Z 683.171,A -85,B 0,C 180,E1 -7905.874,E2 -7905.874} C_VEL
LIN {X 0,Y 462.102,Z 694.858,A -85,B 0,C 180,E1 -7906.589,E2 -7906.589} C_VEL
LIN {X 0,Y 461.667,Z 706.503,A -85,B 0,C 180,E1 -7907.511,E2 -7907.511} C_VEL
LIN {X 0,Y 461.14,Z 717.254,A -85,B 0,C 180,E1 -7908.573,E2 -7908.573} C_VEL
LIN {X 0,Y 460.785,Z 726.233,A -85,B 0,C 180,E1 -7909.676,E2 -7909.676} C_VEL
LIN {X 0,Y 460.347,Z 735.004,A -85,B 0,C 180,E1 -7910.997,E2 -7910.997} C_VEL
LIN {X 0,Y 460.018,Z 742.019,A -85,B 0,C 180,E1 -7912.318,E2 -7912.318} C_VEL
LIN {X 0,Y 459.874,Z 748.397,A -85,B 0,C 180,E1 -7913.859,E2 -7913.859} C_VEL
LIN {X 0,Y 459.66,Z 752.576,A -85,B 0,C 180,E1 -7915.176,E2 -7915.176} C_VEL
LIN {X 0,Y 459.68,Z 755.669,A -85,B 0,C 180,E1 -7916.494,E2 -7916.494} C_VEL
LIN {X 0,Y 459.607,Z 757.195,A -85,B 0,C 180,E1 -7917.371,E2 -7917.371} C_VEL
LIN {X 0,Y 459.523,Z 758.915,A -85,B 0,C 180,E1 -7919.124,E2 -7919.124} C_VEL
LIN {X 0,Y 459.53,Z 759.183,A -85,B 0,C 180,E1 -7920,E2 -7920} C_VEL
LIN {X 0,Y 459.523,Z 759.005,A -85,B 0,C 180,E1 -7920.876,E2 -7920.876} C_VEL
LIN {X 0,Y 459.546,Z 758.412,A -85,B 0,C 180,E1 -7921.753,E2 -7921.753} C_VEL
LIN {X 0,Y 459.607,Z 757.421,A -85,B 0,C 180,E1 -7922.629,E2 -7922.629} C_VEL
LIN {X 0,Y 459.68,Z 756,A -85,B 0,C 180,E1 -7923.506,E2 -7923.506} C_VEL
LIN {X 0,Y 459.656,Z 753.027,A -85,B 0,C 180,E1 -7924.824,E2 -7924.824} C_VEL
LIN {X 0,Y 459.861,Z 748.967,A -85,B 0,C 180,E1 -7926.141,E2 -7926.141} C_VEL
LIN {X 0,Y 460.022,Z 742.7,A -85,B 0,C 180,E1 -7927.682,E2 -7927.682} C_VEL
LIN {X 0,Y 460.351,Z 735.86,A -85,B 0,C 180,E1 -7929.003,E2 -7929.003} C_VEL
LIN {X 0,Y 460.75,Z 727.259,A -85,B 0,C 180,E1 -7930.325,E2 -7930.325} C_VEL
LIN {X 0,Y 461.141,Z 718.442,A -85,B 0,C 180,E1 -7931.427,E2 -7931.427} C_VEL
LIN {X 0,Y 461.658,Z 707.996,A -85,B 0,C 180,E1 -7932.485,E2 -7932.485} C_VEL
LIN {X 0,Y 462.113,Z 696.533,A -85,B 0,C 180,E1 -7933.411,E2 -7933.411} C_VEL
LIN {X 0,Y 462.505,Z 684.28,A -85,B 0,C 180,E1 -7934.184,E2 -7934.184} C_VEL
LIN {X 0,Y 462.979,Z 671.293,A -85,B 0,C 180,E1 -7934.786,E2 -7934.786} C_VEL
LIN {X 0,Y 463.296,Z 658.619,A -85,B 0,C 180,E1 -7935.198,E2 -7935.198} C_VEL
LIN {X 0,Y 463.606,Z 628.824,A -85,B 0,C 180,E1 -7935.75,E2 -7935.75} C_VEL
LIN {X 0,Y 464.549,Z 560.432,A -85,B 0,C 180,E1 -7937.001,E2 -7937.001} C_VEL
LIN {X 0,Y 462.312,Z 546.842,A -85,B 0,C 180,E1 -7937.392,E2 -7937.392} C_VEL
LIN {X 0,Y 463.031,Z 524.775,A -85,B 0,C 180,E1 -7940.664,E2 -7940.664} C_VEL
LIN {X 0,Y 463.789,Z 500.995,A -85,B 0,C 180,E1 -7944.151,E2 -7944.151} C_VEL
LIN {X 0,Y 463.794,Z 492.844,A -85,B 0,C 180,E1 -7945.346,E2 -7945.346} C_VEL
LIN {X 0,Y 461.363,Z 481.336,A -85,B 0,C 180,E1 -7947.193,E2 -7947.193} C_VEL
LIN {X 0,Y 460.581,Z 478.241,A -85,B 0,C 180,E1 -7947.7,E2 -7947.7} C_VEL
LIN {X 0,Y 460.539,Z 478.247,A -85,B 0,C 180,E1 -7951.255,E2 -7951.255} C_VEL
LIN {X 0,Y 460.534,Z 478.247,A -85,B 0,C 180,E1 -7954.505,E2 -7954.505} C_VEL
LIN {X 0,Y 460.503,Z 478.246,A -85,B 0,C 180,E1 -7957.623,E2 -7957.623} C_VEL
LIN {X 0,Y 460.544,Z 478.243,A -85,B 0,C 180,E1 -7960.269,E2 -7960.269} C_VEL
LIN {X 0,Y 460.502,Z 478.244,A -85,B 0,C 180,E1 -7963.375,E2 -7963.375} C_VEL
LIN {X 0,Y 460.511,Z 478.248,A -85,B 0,C 180,E1 -7966.626,E2 -7966.626} C_VEL
LIN {X 0,Y 460.545,Z 478.241,A -85,B 0,C 180,E1 -7969.73,E2 -7969.73} C_VEL
LIN {X 0,Y 460.529,Z 478.245,A -85,B 0,C 180,E1 -7972.519,E2 -7972.519} C_VEL
LIN {X 0,Y 460.55,Z 478.241,A -85,B 0,C 180,E1 -7975.624,E2 -7975.624} C_VEL
LIN {X 0,Y 460.539,Z 478.245,A -85,B 0,C 180,E1 -7978.745,E2 -7978.745} C_VEL
LIN {X 0,Y 460.613,Z 478.422,A -85,B 0,C 180,E1 -7982.161,E2 -7982.161} C_VEL
LIN {X 0,Y 464.18,Z 493.393,A -85,B 0,C 180,E1 -7984.677,E2 -7984.677} C_VEL
LIN {X 0,Y 464.955,Z 497.373,A -85,B 0,C 180,E1 -7985.319,E2 -7985.319} C_VEL
LIN {X 0,Y 463.709,Z 518.756,A -85,B 0,C 180,E1 -7988.436,E2 -7988.436} C_VEL
LIN {X 0,Y 463.37,Z 525.001,A -85,B 0,C 180,E1 -7989.338,E2 -7989.338} C_VEL
LIN {X 0,Y 466.22,Z 544.011,A -85,B 0,C 180,E1 -7989.799,E2 -7989.799} C_VEL
LIN {X 0,Y 464.6,Z 662.902,A -85,B 0,C 180,E1 -7991.821,E2 -7991.821} C_VEL
LIN {X 0,Y 464.175,Z 676.952,A -85,B 0,C 180,E1 -7992.231,E2 -7992.231} C_VEL
LIN {X 0,Y 463.773,Z 689.85,A -85,B 0,C 180,E1 -7992.771,E2 -7992.771} C_VEL
LIN {X 0,Y 463.263,Z 702.659,A -85,B 0,C 180,E1 -7993.474,E2 -7993.474} C_VEL
LIN {X 0,Y 462.558,Z 715.346,A -85,B 0,C 180,E1 -7994.354,E2 -7994.354} C_VEL
LIN {X 0,Y 461.973,Z 726.923,A -85,B 0,C 180,E1 -7995.35,E2 -7995.35} C_VEL
LIN {X 0,Y 461.299,Z 738.516,A -85,B 0,C 180,E1 -7996.565,E2 -7996.565} C_VEL
LIN {X 0,Y 460.862,Z 748.819,A -85,B 0,C 180,E1 -7997.896,E2 -7997.896} C_VEL
LIN {X 0,Y 460.422,Z 757.331,A -85,B 0,C 180,E1 -7999.223,E2 -7999.223} C_VEL
LIN {X 0,Y 460.048,Z 765.439,A -85,B 0,C 180,E1 -8000.77,E2 -8000.77} C_VEL
LIN {X 0,Y 459.807,Z 771.121,A -85,B 0,C 180,E1 -8002.093,E2 -8002.093} C_VEL
LIN {X 0,Y 459.712,Z 776.227,A -85,B 0,C 180,E1 -8003.57,E2 -8003.57} C_VEL
LIN {X 0,Y 459.648,Z 779.393,A -85,B 0,C 180,E1 -8004.736,E2 -8004.736} C_VEL
LIN {X 0,Y 459.576,Z 782.934,A -85,B 0,C 180,E1 -8006.493,E2 -8006.493} C_VEL
LIN {X 0,Y 459.539,Z 785.027,A -85,B 0,C 180,E1 -8008.247,E2 -8008.247} C_VEL
LIN {X 0,Y 459.528,Z 785.714,A -85,B 0,C 180,E1 -8010,E2 -8010} C_VEL
LIN {X 0,Y 459.539,Z 784.988,A -85,B 0,C 180,E1 -8011.753,E2 -8011.753} C_VEL
LIN {X 0,Y 459.576,Z 782.851,A -85,B 0,C 180,E1 -8013.507,E2 -8013.507} C_VEL
LIN {X 0,Y 459.648,Z 779.251,A -85,B 0,C 180,E1 -8015.264,E2 -8015.264} C_VEL
LIN {X 0,Y 459.713,Z 776.035,A -85,B 0,C 180,E1 -8016.431,E2 -8016.431} C_VEL
LIN {X 0,Y 459.798,Z 770.872,A -85,B 0,C 180,E1 -8017.907,E2 -8017.907} C_VEL
LIN {X 0,Y 460.079,Z 764.087,A -85,B 0,C 180,E1 -8019.452,E2 -8019.452} C_VEL
LIN {X 0,Y 460.451,Z 755.589,A -85,B 0,C 180,E1 -8020.999,E2 -8020.999} C_VEL
LIN {X 0,Y 460.91,Z 745.687,A -85,B 0,C 180,E1 -8022.459,E2 -8022.459} C_VEL
LIN {X 0,Y 461.435,Z 734.856,A -85,B 0,C 180,E1 -8023.768,E2 -8023.768} C_VEL
LIN {X 0,Y 462.001,Z 723.69,A -85,B 0,C 180,E1 -8024.875,E2 -8024.875} C_VEL
LIN {X 0,Y 462.654,Z 711.412,A -85,B 0,C 180,E1 -8025.869,E2 -8025.869} C_VEL
LIN {X 0,Y 463.228,Z 699.594,A -85,B 0,C 180,E1 -8026.641,E2 -8026.641} C_VEL
LIN {X 0,Y 463.786,Z 685.985,A -85,B 0,C 180,E1 -8027.336,E2 -8027.336} C_VEL
LIN {X 0,Y 464.253,Z 671.403,A -85,B 0,C 180,E1 -8027.88,E2 -8027.88} C_VEL
LIN {X 0,Y 464.6,Z 656.733,A -85,B 0,C 180,E1 -8028.237,E2 -8028.237} C_VEL
LIN {X 0,Y 466.036,Z 555.786,A -85,B 0,C 180,E1 -8029.984,E2 -8029.984} C_VEL
LIN {X 0,Y 466.13,Z 542.118,A -85,B 0,C 180,E1 -8030.239,E2 -8030.239} C_VEL
LIN {X 0,Y 463.575,Z 525.849,A -85,B 0,C 180,E1 -8030.694,E2 -8030.694} C_VEL
LIN {X 0,Y 465.206,Z 503.635,A -85,B 0,C 180,E1 -8034.073,E2 -8034.073} C_VEL
LIN {X 0,Y 465.569,Z 498.956,A -85,B 0,C 180,E1 -8034.809,E2 -8034.809} C_VEL
LIN {X 0,Y 463.435,Z 488.694,A -85,B 0,C 180,E1 -8036.704,E2 -8036.704} C_VEL
LIN {X 0,Y 460.556,Z 478.244,A -85,B 0,C 180,E1 -8038.855,E2 -8038.855} C_VEL
LIN {X 0,Y 460.534,Z 478.245,A -85,B 0,C 180,E1 -8042.284,E2 -8042.284} C_VEL
LIN {X 0,Y 460.512,Z 478.25,A -85,B 0,C 180,E1 -8045.446,E2 -8045.446} C_VEL
LIN {X 0,Y 460.547,Z 478.244,A -85,B 0,C 180,E1 -8048.898,E2 -8048.898} C_VEL
LIN {X 0,Y 460.526,Z 478.243,A -85,B 0,C 180,E1 -8052.181,E2 -8052.181} C_VEL
LIN {X 0,Y 460.52,Z 478.246,A -85,B 0,C 180,E1 -8055.412,E2 -8055.412} C_VEL
LIN {X 0,Y 460.535,Z 478.244,A -85,B 0,C 180,E1 -8058.398,E2 -8058.398} C_VEL
LIN {X 0,Y 460.53,Z 478.246,A -85,B 0,C 180,E1 -8061.267,E2 -8061.267} C_VEL
LIN {X 0,Y 460.514,Z 478.249,A -85,B 0,C 180,E1 -8064.555,E2 -8064.555} C_VEL
LIN {X 0,Y 460.535,Z 478.244,A -85,B 0,C 180,E1 -8067.716,E2 -8067.716} C_VEL
LIN {X 0,Y 460.544,Z 478.25,A -85,B 0,C 180,E1 -8070.769,E2 -8070.769} C_VEL
LIN {X 0,Y 460.585,Z 478.371,A -85,B 0,C 180,E1 -8071.912,E2 -8071.912} C_VEL
LIN {X 0,Y 462.902,Z 487.255,A -85,B 0,C 180,E1 -8073.877,E2 -8073.877} C_VEL
LIN {X 0,Y 464.845,Z 497.226,A -85,B 0,C 180,E1 -8075.907,E2 -8075.907} C_VEL
LIN {X 0,Y 463.767,Z 511.628,A -85,B 0,C 180,E1 -8078.439,E2 -8078.439} C_VEL
LIN {X 0,Y 462.717,Z 530.25,A -85,B 0,C 180,E1 -8081.629,E2 -8081.629} C_VEL
LIN {X 0,Y 462.204,Z 540.565,A -85,B 0,C 180,E1 -8083.325,E2 -8083.325} C_VEL
LIN {X 0,Y 465.175,Z 557.817,A -85,B 0,C 180,E1 -8083.829,E2 -8083.829} C_VEL
LIN {X 0,Y 464.933,Z 575.785,A -85,B 0,C 180,E1 -8084.191,E2 -8084.191} C_VEL
LIN {X 0,Y 463.549,Z 654.074,A -85,B 0,C 180,E1 -8085.709,E2 -8085.709} C_VEL
LIN {X 0,Y 463.222,Z 667.412,A -85,B 0,C 180,E1 -8086.145,E2 -8086.145} C_VEL
LIN {X 0,Y 462.834,Z 679.975,A -85,B 0,C 180,E1 -8086.735,E2 -8086.735} C_VEL
LIN {X 0,Y 462.382,Z 692.128,A -85,B 0,C 180,E1 -8087.491,E2 -8087.491} C_VEL
LIN {X 0,Y 461.814,Z 703.288,A -85,B 0,C 180,E1 -8088.367,E2 -8088.367} C_VEL
LIN {X 0,Y 461.359,Z 712.369,A -85,B 0,C 180,E1 -8089.245,E2 -8089.245} C_VEL
LIN {X 0,Y 460.982,Z 721.708,A -85,B 0,C 180,E1 -8090.346,E2 -8090.346} C_VEL
LIN {X 0,Y 460.468,Z 730.789,A -85,B 0,C 180,E1 -8091.663,E2 -8091.663} C_VEL
LIN {X 0,Y 460.178,Z 738.104,A -85,B 0,C 180,E1 -8092.982,E2 -8092.982} C_VEL
LIN {X 0,Y 459.935,Z 743.938,A -85,B 0,C 180,E1 -8094.3,E2 -8094.3} C_VEL
LIN {X 0,Y 459.816,Z 748.529,A -85,B 0,C 180,E1 -8095.617,E2 -8095.617} C_VEL
LIN {X 0,Y 459.754,Z 750.942,A -85,B 0,C 180,E1 -8096.494,E2 -8096.494} C_VEL
LIN {X 0,Y 459.654,Z 752.917,A -85,B 0,C 180,E1 -8097.371,E2 -8097.371} C_VEL
LIN {X 0,Y 459.581,Z 754.463,A -85,B 0,C 180,E1 -8098.247,E2 -8098.247} C_VEL
LIN {X 0,Y 459.555,Z 755.538,A -85,B 0,C 180,E1 -8099.124,E2 -8099.124} C_VEL
LIN {X 0,Y 459.531,Z 756.207,A -85,B 0,C 180,E1 -8100,E2 -8100} C_VEL
LIN {X 0,Y 459.523,Z 756.478,A -85,B 0,C 180,E1 -8100.876,E2 -8100.876} C_VEL
LIN {X 0,Y 459.546,Z 756.342,A -85,B 0,C 180,E1 -8101.753,E2 -8101.753} C_VEL
LIN {X 0,Y 459.602,Z 755.757,A -85,B 0,C 180,E1 -8102.629,E2 -8102.629} C_VEL
LIN {X 0,Y 459.642,Z 754.77,A -85,B 0,C 180,E1 -8103.506,E2 -8103.506} C_VEL
LIN {X 0,Y 459.596,Z 753.378,A -85,B 0,C 180,E1 -8104.385,E2 -8104.385} C_VEL
LIN {X 0,Y 459.739,Z 750.441,A -85,B 0,C 180,E1 -8105.703,E2 -8105.703} C_VEL
LIN {X 0,Y 459.792,Z 746.448,A -85,B 0,C 180,E1 -8107.024,E2 -8107.024} C_VEL
LIN {X 0,Y 460.024,Z 740.294,A -85,B 0,C 180,E1 -8108.566,E2 -8108.566} C_VEL
LIN {X 0,Y 460.324,Z 733.532,A -85,B 0,C 180,E1 -8109.89,E2 -8109.89} C_VEL
LIN {X 0,Y 460.743,Z 725.125,A -85,B 0,C 180,E1 -8111.215,E2 -8111.215} C_VEL
LIN {X 0,Y 461.105,Z 716.521,A -85,B 0,C 180,E1 -8112.321,E2 -8112.321} C_VEL
LIN {X 0,Y 461.562,Z 705.896,A -85,B 0,C 180,E1 -8113.427,E2 -8113.427} C_VEL
LIN {X 0,Y 462.189,Z 693.964,A -85,B 0,C 180,E1 -8114.418,E2 -8114.418} C_VEL
LIN {X 0,Y 462.625,Z 682.025,A -85,B 0,C 180,E1 -8115.192,E2 -8115.192} C_VEL
LIN {X 0,Y 463.056,Z 668.469,A -85,B 0,C 180,E1 -8115.854,E2 -8115.854} C_VEL
LIN {X 0,Y 463.419,Z 655.448,A -85,B 0,C 180,E1 -8116.294,E2 -8116.294} C_VEL
LIN {X 0,Y 463.708,Z 637.43,A -85,B 0,C 180,E1 -8116.651,E2 -8116.651} C_VEL
LIN {X 0,Y 464.658,Z 557.695,A -85,B 0,C 180,E1 -8118.063,E2 -8118.063} C_VEL
LIN {X 0,Y 461.935,Z 540.872,A -85,B 0,C 180,E1 -8118.489,E2 -8118.489} C_VEL
LIN {X 0,Y 462.664,Z 524.699,A -85,B 0,C 180,E1 -8121.147,E2 -8121.147} C_VEL
LIN {X 0,Y 463.611,Z 506.593,A -85,B 0,C 180,E1 -8124.161,E2 -8124.161} C_VEL
LIN {X 0,Y 464.198,Z 495.403,A -85,B 0,C 180,E1 -8126.044,E2 -8126.044} C_VEL
LIN {X 0,Y 461.905,Z 484.075,A -85,B 0,C 180,E1 -8128.143,E2 -8128.143} C_VEL
LIN {X 0,Y 460.549,Z 478.245,A -85,B 0,C 180,E1 -8129.29,E2 -8129.29} C_VEL
LIN {X 0,Y 460.534,Z 478.244,A -85,B 0,C 180,E1 -8132.284,E2 -8132.284} C_VEL
LIN {X 0,Y 460.514,Z 478.248,A -85,B 0,C 180,E1 -8135.445,E2 -8135.445} C_VEL
LIN {X 0,Y 460.547,Z 478.238,A -85,B 0,C 180,E1 -8138.898,E2 -8138.898} C_VEL
LIN {X 0,Y 460.525,Z 478.242,A -85,B 0,C 180,E1 -8142.181,E2 -8142.181} C_VEL
LIN {X 0,Y 460.516,Z 478.247,A -85,B 0,C 180,E1 -8145.411,E2 -8145.411} C_VEL
LIN {X 0,Y 460.534,Z 478.239,A -85,B 0,C 180,E1 -8148.397,E2 -8148.397} C_VEL
LIN {X 0,Y 460.521,Z 478.245,A -85,B 0,C 180,E1 -8151.266,E2 -8151.266} C_VEL
LIN {X 0,Y 460.512,Z 478.242,A -85,B 0,C 180,E1 -8154.554,E2 -8154.554} C_VEL
LIN {X 0,Y 460.533,Z 478.245,A -85,B 0,C 180,E1 -8157.715,E2 -8157.715} C_VEL
LIN {X 0,Y 460.521,Z 478.241,A -85,B 0,C 180,E1 -8160.257,E2 -8160.257} C_VEL
LIN {X 0,Y 459.886,Z 478.323,A -85,B 0,C 180,E1 -8160.987,E2 -8160.987} C_VEL
LIN {X 0,Y 457.043,Z 478.677,A -85,B 0,C 180,E1 -8162.172,E2 -8162.172} C_VEL
LIN {X 0,Y 454.626,Z 478.98,A -85,B 0,C 180,E1 -8163.128,E2 -8163.128} C_VEL
LIN {X 0,Y 453.598,Z 479.108,A -85,B 0,C 180,E1 -8163.867,E2 -8163.867} C_VEL
LIN {X 0,Y 453.521,Z 479.114,A -85,B 0,C 180,E1 -8164.117,E2 -8164.117} C_VEL
LIN {X 0,Y 453.481,Z 479.122,A -85,B 0,C 180,E1 -8167.204,E2 -8167.204} C_VEL
LIN {X 0,Y 453.507,Z 479.116,A -85,B 0,C 180,E1 -8170.066,E2 -8170.066} C_VEL
LIN {X 0,Y 453.509,Z 479.115,A -85,B 0,C 180,E1 -8172.876,E2 -8172.876} C_VEL
LIN {X 0,Y 453.518,Z 479.119,A -85,B 0,C 180,E1 -8175.644,E2 -8175.644} C_VEL
LIN {X 0,Y 453.562,Z 479.108,A -85,B 0,C 180,E1 -8178.379,E2 -8178.379} C_VEL
LIN {X 0,Y 453.654,Z 479.098,A -85,B 0,C 180,E1 -8181.985,E2 -8181.985} C_VEL
LIN {X 0,Y 453.673,Z 479.094,A -85,B 0,C 180,E1 -8184.667,E2 -8184.667} C_VEL
LIN {X 0,Y 453.767,Z 479.089,A -85,B 0,C 180,E1 -8187.337,E2 -8187.337} C_VEL
LIN {X 0,Y 453.826,Z 479.076,A -85,B 0,C 180,E1 -8190,E2 -8190} C_VEL
LIN {X 0,Y 453.768,Z 479.082,A -85,B 0,C 180,E1 -8192.663,E2 -8192.663} C_VEL
LIN {X 0,Y 453.671,Z 479.094,A -85,B 0,C 180,E1 -8196.225,E2 -8196.225} C_VEL
LIN {X 0,Y 453.594,Z 479.106,A -85,B 0,C 180,E1 -8198.913,E2 -8198.913} C_VEL
LIN {X 0,Y 453.565,Z 479.107,A -85,B 0,C 180,E1 -8202.529,E2 -8202.529} C_VEL
LIN {X 0,Y 453.546,Z 479.11,A -85,B 0,C 180,E1 -8206.196,E2 -8206.196} C_VEL
LIN {X 0,Y 453.522,Z 479.116,A -85,B 0,C 180,E1 -8209.041,E2 -8209.041} C_VEL
LIN {X 0,Y 453.479,Z 479.121,A -85,B 0,C 180,E1 -8211.836,E2 -8211.836} C_VEL
LIN {X 0,Y 453.516,Z 479.114,A -85,B 0,C 180,E1 -8214.734,E2 -8214.734} C_VEL
LIN {X 0,Y 453.539,Z 479.112,A -85,B 0,C 180,E1 -8217.961,E2 -8217.961} C_VEL
LIN {X 0,Y 453.468,Z 479.125,A -85,B 0,C 180,E1 -8221.525,E2 -8221.525} C_VEL
LIN {X 0,Y 453.489,Z 479.118,A -85,B 0,C 180,E1 -8224.777,E2 -8224.777} C_VEL
LIN {X 0,Y 453.466,Z 479.12,A -85,B 0,C 180,E1 -8228.312,E2 -8228.312} C_VEL
LIN {X 0,Y 453.496,Z 479.117,A -85,B 0,C 180,E1 -8230.609,E2 -8230.609} C_VEL
LIN {X 0,Y 453.466,Z 479.127,A -85,B 0,C 180,E1 -8233.245,E2 -8233.245} C_VEL
LIN {X 0,Y 453.468,Z 479.122,A -85,B 0,C 180,E1 -8235.779,E2 -8235.779} C_VEL
LIN {X 0,Y 453.481,Z 479.118,A -85,B 0,C 180,E1 -8238.209,E2 -8238.209} C_VEL
LIN {X 0,Y 453.496,Z 479.118,A -85,B 0,C 180,E1 -8240.793,E2 -8240.793} C_VEL
LIN {X 0,Y 453.456,Z 479.122,A -85,B 0,C 180,E1 -8243.917,E2 -8243.917} C_VEL
LIN {X 0,Y 453.485,Z 479.124,A -85,B 0,C 180,E1 -8247.151,E2 -8247.151} C_VEL
LIN {X 0,Y 453.477,Z 479.119,A -85,B 0,C 180,E1 -8250.268,E2 -8250.268} C_VEL
LIN {X 0,Y 453.554,Z 479.247,A -85,B 0,C 180,E1 -8252.083,E2 -8252.083} C_VEL
LIN {X 0,Y 456.603,Z 493.448,A -85,B 0,C 180,E1 -8254.471,E2 -8254.471} C_VEL
LIN {X 0,Y 456.914,Z 497.816,A -85,B 0,C 180,E1 -8255.163,E2 -8255.163} C_VEL
LIN {X 0,Y 456.165,Z 517.019,A -85,B 0,C 180,E1 -8258.109,E2 -8258.109} C_VEL
LIN {X 0,Y 455.485,Z 536.501,A -85,B 0,C 180,E1 -8261.094,E2 -8261.094} C_VEL
LIN {X 0,Y 455.157,Z 546.455,A -85,B 0,C 180,E1 -8262.594,E2 -8262.594} C_VEL
LIN {X 0,Y 457.554,Z 562.988,A -85,B 0,C 180,E1 -8262.984,E2 -8262.984} C_VEL
LIN {X 0,Y 456.439,Z 656.697,A -85,B 0,C 180,E1 -8264.654,E2 -8264.654} C_VEL
LIN {X 0,Y 456.076,Z 669.342,A -85,B 0,C 180,E1 -8265.042,E2 -8265.042} C_VEL
LIN {X 0,Y 455.615,Z 682.721,A -85,B 0,C 180,E1 -8265.654,E2 -8265.654} C_VEL
LIN {X 0,Y 455.184,Z 694.567,A -85,B 0,C 180,E1 -8266.381,E2 -8266.381} C_VEL
LIN {X 0,Y 454.685,Z 706.522,A -85,B 0,C 180,E1 -8267.335,E2 -8267.335} C_VEL
LIN {X 0,Y 454.159,Z 717.145,A -85,B 0,C 180,E1 -8268.395,E2 -8268.395} C_VEL
LIN {X 0,Y 453.774,Z 726.191,A -85,B 0,C 180,E1 -8269.515,E2 -8269.515} C_VEL
LIN {X 0,Y 453.32,Z 735.01,A -85,B 0,C 180,E1 -8270.856,E2 -8270.856} C_VEL
LIN {X 0,Y 452.968,Z 742.079,A -85,B 0,C 180,E1 -8272.197,E2 -8272.197} C_VEL
LIN {X 0,Y 452.804,Z 748.496,A -85,B 0,C 180,E1 -8273.763,E2 -8273.763} C_VEL
LIN {X 0,Y 452.594,Z 752.705,A -85,B 0,C 180,E1 -8275.101,E2 -8275.101} C_VEL
LIN {X 0,Y 452.581,Z 755.823,A -85,B 0,C 180,E1 -8276.439,E2 -8276.439} C_VEL
LIN {X 0,Y 452.533,Z 757.362,A -85,B 0,C 180,E1 -8277.33,E2 -8277.33} C_VEL
LIN {X 0,Y 452.461,Z 758.432,A -85,B 0,C 180,E1 -8278.22,E2 -8278.22} C_VEL
LIN {X 0,Y 452.43,Z 759.102,A -85,B 0,C 180,E1 -8279.11,E2 -8279.11} C_VEL
LIN {X 0,Y 452.434,Z 759.376,A -85,B 0,C 180,E1 -8280,E2 -8280} C_VEL
LIN {X 0,Y 452.43,Z 759.203,A -85,B 0,C 180,E1 -8280.89,E2 -8280.89} C_VEL
LIN {X 0,Y 452.461,Z 758.611,A -85,B 0,C 180,E1 -8281.78,E2 -8281.78} C_VEL
LIN {X 0,Y 452.533,Z 757.622,A -85,B 0,C 180,E1 -8282.67,E2 -8282.67} C_VEL
LIN {X 0,Y 452.596,Z 756.203,A -85,B 0,C 180,E1 -8283.561,E2 -8283.561} C_VEL
LIN {X 0,Y 452.59,Z 753.233,A -85,B 0,C 180,E1 -8284.899,E2 -8284.899} C_VEL
LIN {X 0,Y 452.802,Z 749.175,A -85,B 0,C 180,E1 -8286.237,E2 -8286.237} C_VEL
LIN {X 0,Y 452.988,Z 742.917,A -85,B 0,C 180,E1 -8287.802,E2 -8287.802} C_VEL
LIN {X 0,Y 453.339,Z 736.06,A -85,B 0,C 180,E1 -8289.143,E2 -8289.143} C_VEL
LIN {X 0,Y 453.754,Z 727.439,A -85,B 0,C 180,E1 -8290.486,E2 -8290.486} C_VEL
LIN {X 0,Y 454.246,Z 717.627,A -85,B 0,C 180,E1 -8291.716,E2 -8291.716} C_VEL
LIN {X 0,Y 454.796,Z 706.554,A -85,B 0,C 180,E1 -8292.818,E2 -8292.818} C_VEL
LIN {X 0,Y 455.269,Z 695.082,A -85,B 0,C 180,E1 -8293.73,E2 -8293.73} C_VEL
LIN {X 0,Y 455.665,Z 683.322,A -85,B 0,C 180,E1 -8294.458,E2 -8294.458} C_VEL
LIN {X 0,Y 456.177,Z 670.075,A -85,B 0,C 180,E1 -8295.069,E2 -8295.069} C_VEL
LIN {X 0,Y 456.496,Z 657.687,A -85,B 0,C 180,E1 -8295.458,E2 -8295.458} C_VEL
LIN {X 0,Y 457.831,Z 561.183,A -85,B 0,C 180,E1 -8297.281,E2 -8297.281} C_VEL
LIN {X 0,Y 455.483,Z 547.078,A -85,B 0,C 180,E1 -8297.706,E2 -8297.706} C_VEL
LIN {X 0,Y 456.202,Z 525.114,A -85,B 0,C 180,E1 -8300.988,E2 -8300.988} C_VEL
LIN {X 0,Y 456.782,Z 507.718,A -85,B 0,C 180,E1 -8303.58,E2 -8303.58} C_VEL
LIN {X 0,Y 457.171,Z 496.052,A -85,B 0,C 180,E1 -8305.297,E2 -8305.297} C_VEL
LIN {X 0,Y 455.413,Z 486.488,A -85,B 0,C 180,E1 -8306.832,E2 -8306.832} C_VEL
LIN {X 0,Y 453.538,Z 479.118,A -85,B 0,C 180,E1 -8308.08,E2 -8308.08} C_VEL
LIN {X 0,Y 453.468,Z 479.127,A -85,B 0,C 180,E1 -8311.525,E2 -8311.525} C_VEL
LIN {X 0,Y 453.49,Z 479.124,A -85,B 0,C 180,E1 -8314.777,E2 -8314.777} C_VEL
LIN {X 0,Y 453.467,Z 479.127,A -85,B 0,C 180,E1 -8318.311,E2 -8318.311} C_VEL
LIN {X 0,Y 453.496,Z 479.121,A -85,B 0,C 180,E1 -8320.609,E2 -8320.609} C_VEL
LIN {X 0,Y 453.458,Z 479.123,A -85,B 0,C 180,E1 -8323.244,E2 -8323.244} C_VEL
LIN {X 0,Y 453.475,Z 479.12,A -85,B 0,C 180,E1 -8325.78,E2 -8325.78} C_VEL
LIN {X 0,Y 453.484,Z 479.124,A -85,B 0,C 180,E1 -8328.21,E2 -8328.21} C_VEL
LIN {X 0,Y 453.517,Z 479.117,A -85,B 0,C 180,E1 -8330.79,E2 -8330.79} C_VEL
LIN {X 0,Y 453.459,Z 479.126,A -85,B 0,C 180,E1 -8333.917,E2 -8333.917} C_VEL
LIN {X 0,Y 453.485,Z 479.121,A -85,B 0,C 180,E1 -8337.151,E2 -8337.151} C_VEL
LIN {X 0,Y 453.516,Z 479.121,A -85,B 0,C 180,E1 -8340.271,E2 -8340.271} C_VEL
LIN {X 0,Y 453.537,Z 479.176,A -85,B 0,C 180,E1 -8341.839,E2 -8341.839} C_VEL
LIN {X 0,Y 457.302,Z 494.845,A -85,B 0,C 180,E1 -8344.512,E2 -8344.512} C_VEL
LIN {X 0,Y 458.104,Z 499.834,A -85,B 0,C 180,E1 -8345.322,E2 -8345.322} C_VEL
LIN {X 0,Y 456.709,Z 521.94,A -85,B 0,C 180,E1 -8348.587,E2 -8348.587} C_VEL
LIN {X 0,Y 456.506,Z 525.118,A -85,B 0,C 180,E1 -8349.05,E2 -8349.05} C_VEL
LIN {X 0,Y 459.493,Z 543.848,A -85,B 0,C 180,E1 -8349.524,E2 -8349.524} C_VEL
LIN {X 0,Y 457.783,Z 661.937,A -85,B 0,C 180,E1 -8351.569,E2 -8351.569} C_VEL
LIN {X 0,Y 457.349,Z 676.239,A -85,B 0,C 180,E1 -8351.985,E2 -8351.985} C_VEL
LIN {X 0,Y 456.865,Z 690.421,A -85,B 0,C 180,E1 -8352.589,E2 -8352.589} C_VEL
LIN {X 0,Y 456.32,Z 703.503,A -85,B 0,C 180,E1 -8353.33,E2 -8353.33} C_VEL
LIN {X 0,Y 455.562,Z 715.999,A -85,B 0,C 180,E1 -8354.222,E2 -8354.222} C_VEL
LIN {X 0,Y 454.965,Z 727.439,A -85,B 0,C 180,E1 -8355.233,E2 -8355.233} C_VEL
LIN {X 0,Y 454.322,Z 737.936,A -85,B 0,C 180,E1 -8356.355,E2 -8356.355} C_VEL
LIN {X 0,Y 453.865,Z 748.351,A -85,B 0,C 180,E1 -8357.707,E2 -8357.707} C_VEL
LIN {X 0,Y 453.38,Z 756.923,A -85,B 0,C 180,E1 -8359.054,E2 -8359.054} C_VEL
LIN {X 0,Y 452.986,Z 765.083,A -85,B 0,C 180,E1 -8360.624,E2 -8360.624} C_VEL
LIN {X 0,Y 452.737,Z 770.804,A -85,B 0,C 180,E1 -8361.969,E2 -8361.969} C_VEL
LIN {X 0,Y 452.604,Z 776.344,A -85,B 0,C 180,E1 -8363.611,E2 -8363.611} C_VEL
LIN {X 0,Y 452.563,Z 779.125,A -85,B 0,C 180,E1 -8364.654,E2 -8364.654} C_VEL
LIN {X 0,Y 452.473,Z 782.686,A -85,B 0,C 180,E1 -8366.438,E2 -8366.438} C_VEL
LIN {X 0,Y 452.504,Z 783.919,A -85,B 0,C 180,E1 -8367.329,E2 -8367.329} C_VEL
LIN {X 0,Y 452.428,Z 785.317,A -85,B 0,C 180,E1 -8369.11,E2 -8369.11} C_VEL
LIN {X 0,Y 452.428,Z 785.302,A -85,B 0,C 180,E1 -8370.89,E2 -8370.89} C_VEL
LIN {X 0,Y 452.504,Z 783.868,A -85,B 0,C 180,E1 -8372.671,E2 -8372.671} C_VEL
LIN {X 0,Y 452.474,Z 780.999,A -85,B 0,C 180,E1 -8374.454,E2 -8374.454} C_VEL
LIN {X 0,Y 452.557,Z 777.893,A -85,B 0,C 180,E1 -8375.794,E2 -8375.794} C_VEL
LIN {X 0,Y 452.654,Z 773.818,A -85,B 0,C 180,E1 -8377.135,E2 -8377.135} C_VEL
LIN {X 0,Y 452.806,Z 768.782,A -85,B 0,C 180,E1 -8378.479,E2 -8378.479} C_VEL
LIN {X 0,Y 453.093,Z 761.51,A -85,B 0,C 180,E1 -8380.05,E2 -8380.05} C_VEL
LIN {X 0,Y 453.519,Z 753.869,A -85,B 0,C 180,E1 -8381.396,E2 -8381.396} C_VEL
LIN {X 0,Y 453.944,Z 744.671,A -85,B 0,C 180,E1 -8382.742,E2 -8382.742} C_VEL
LIN {X 0,Y 454.522,Z 733.46,A -85,B 0,C 180,E1 -8384.095,E2 -8384.095} C_VEL
LIN {X 0,Y 455.128,Z 722.029,A -85,B 0,C 180,E1 -8385.219,E2 -8385.219} C_VEL
LIN {X 0,Y 455.881,Z 709.336,A -85,B 0,C 180,E1 -8386.226,E2 -8386.226} C_VEL
LIN {X 0,Y 456.553,Z 695.494,A -85,B 0,C 180,E1 -8387.096,E2 -8387.096} C_VEL
LIN {X 0,Y 457.15,Z 681.296,A -85,B 0,C 180,E1 -8387.776,E2 -8387.776} C_VEL
LIN {X 0,Y 457.594,Z 667.935,A -85,B 0,C 180,E1 -8388.236,E2 -8388.236} C_VEL
LIN {X 0,Y 457.913,Z 652.539,A -85,B 0,C 180,E1 -8388.57,E2 -8388.57} C_VEL
LIN {X 0,Y 459.311,Z 559.839,A -85,B 0,C 180,E1 -8390.221,E2 -8390.221} C_VEL
LIN {X 0,Y 459.503,Z 543.06,A -85,B 0,C 180,E1 -8390.541,E2 -8390.541} C_VEL
LIN {X 0,Y 456.884,Z 526.684,A -85,B 0,C 180,E1 -8391.006,E2 -8391.006} C_VEL
LIN {X 0,Y 456.794,Z 526.13,A -85,B 0,C 180,E1 -8391.032,E2 -8391.032} C_VEL
LIN {X 0,Y 458.588,Z 504.202,A -85,B 0,C 180,E1 -8394.443,E2 -8394.443} C_VEL
LIN {X 0,Y 458.805,Z 500.46,A -85,B 0,C 180,E1 -8395.056,E2 -8395.056} C_VEL
LIN {X 0,Y 456.555,Z 490.006,A -85,B 0,C 180,E1 -8397.061,E2 -8397.061} C_VEL
LIN {X 0,Y 453.509,Z 479.125,A -85,B 0,C 180,E1 -8399.395,E2 -8399.395} C_VEL
LIN {X 0,Y 453.485,Z 479.124,A -85,B 0,C 180,E1 -8402.849,E2 -8402.849} C_VEL
LIN {X 0,Y 453.456,Z 479.127,A -85,B 0,C 180,E1 -8406.083,E2 -8406.083} C_VEL
LIN {X 0,Y 453.508,Z 479.122,A -85,B 0,C 180,E1 -8409.448,E2 -8409.448} C_VEL
LIN {X 0,Y 453.471,Z 479.126,A -85,B 0,C 180,E1 -8412.994,E2 -8412.994} C_VEL
LIN {X 0,Y 453.469,Z 479.124,A -85,B 0,C 180,E1 -8415.779,E2 -8415.779} C_VEL
LIN {X 0,Y 453.482,Z 479.121,A -85,B 0,C 180,E1 -8418.209,E2 -8418.209} C_VEL
LIN {X 0,Y 453.513,Z 479.122,A -85,B 0,C 180,E1 -8420.791,E2 -8420.791} C_VEL
LIN {X 0,Y 453.458,Z 479.126,A -85,B 0,C 180,E1 -8423.917,E2 -8423.917} C_VEL
LIN {X 0,Y 453.486,Z 479.125,A -85,B 0,C 180,E1 -8427.151,E2 -8427.151} C_VEL
LIN {X 0,Y 453.479,Z 479.128,A -85,B 0,C 180,E1 -8430.269,E2 -8430.269} C_VEL
LIN {X 0,Y 453.519,Z 479.324,A -85,B 0,C 180,E1 -8431.389,E2 -8431.389} C_VEL
LIN {X 0,Y 455.894,Z 487.945,A -85,B 0,C 180,E1 -8433.396,E2 -8433.396} C_VEL
LIN {X 0,Y 457.937,Z 497.973,A -85,B 0,C 180,E1 -8435.52,E2 -8435.52} C_VEL
LIN {X 0,Y 458.036,Z 500.509,A -85,B 0,C 180,E1 -8436.008,E2 -8436.008} C_VEL
LIN {X 0,Y 456.553,Z 520.08,A -85,B 0,C 180,E1 -8439.491,E2 -8439.491} C_VEL
LIN {X 0,Y 455.551,Z 536.104,A -85,B 0,C 180,E1 -8442.26,E2 -8442.26} C_VEL
LIN {X 0,Y 455.336,Z 540.136,A -85,B 0,C 180,E1 -8442.947,E2 -8442.947} C_VEL
LIN {X 0,Y 458.291,Z 557.006,A -85,B 0,C 180,E1 -8443.48,E2 -8443.48} C_VEL
LIN {X 0,Y 458.66,Z 561.973,A -85,B 0,C 180,E1 -8443.608,E2 -8443.608} C_VEL
LIN {X 0,Y 456.794,Z 653.61,A -85,B 0,C 180,E1 -8445.436,E2 -8445.436} C_VEL
LIN {X 0,Y 456.444,Z 666.922,A -85,B 0,C 180,E1 -8445.876,E2 -8445.876} C_VEL
LIN {X 0,Y 456.031,Z 679.04,A -85,B 0,C 180,E1 -8446.442,E2 -8446.442} C_VEL
LIN {X 0,Y 455.537,Z 691.053,A -85,B 0,C 180,E1 -8447.187,E2 -8447.187} C_VEL
LIN {X 0,Y 454.956,Z 702.395,A -85,B 0,C 180,E1 -8448.076,E2 -8448.076} C_VEL
LIN {X 0,Y 454.408,Z 712.744,A -85,B 0,C 180,E1 -8449.079,E2 -8449.079} C_VEL
LIN {X 0,Y 453.999,Z 722.059,A -85,B 0,C 180,E1 -8450.196,E2 -8450.196} C_VEL
LIN {X 0,Y 453.461,Z 731.139,A -85,B 0,C 180,E1 -8451.533,E2 -8451.533} C_VEL
LIN {X 0,Y 453.136,Z 738.446,A -85,B 0,C 180,E1 -8452.872,E2 -8452.872} C_VEL
LIN {X 0,Y 452.898,Z 744.26,A -85,B 0,C 180,E1 -8454.211,E2 -8454.211} C_VEL
LIN {X 0,Y 452.727,Z 748.827,A -85,B 0,C 180,E1 -8455.548,E2 -8455.548} C_VEL
LIN {X 0,Y 452.695,Z 751.229,A -85,B 0,C 180,E1 -8456.44,E2 -8456.44} C_VEL
LIN {X 0,Y 452.579,Z 753.195,A -85,B 0,C 180,E1 -8457.33,E2 -8457.33} C_VEL
LIN {X 0,Y 452.495,Z 754.728,A -85,B 0,C 180,E1 -8458.22,E2 -8458.22} C_VEL
LIN {X 0,Y 452.46,Z 755.791,A -85,B 0,C 180,E1 -8459.11,E2 -8459.11} C_VEL
LIN {X 0,Y 452.435,Z 756.449,A -85,B 0,C 180,E1 -8460,E2 -8460} C_VEL
LIN {X 0,Y 452.43,Z 756.71,A -85,B 0,C 180,E1 -8460.89,E2 -8460.89} C_VEL
LIN {X 0,Y 452.461,Z 756.557,A -85,B 0,C 180,E1 -8461.78,E2 -8461.78} C_VEL
LIN {X 0,Y 452.527,Z 755.953,A -85,B 0,C 180,E1 -8462.67,E2 -8462.67} C_VEL
LIN {X 0,Y 452.542,Z 754.949,A -85,B 0,C 180,E1 -8463.562,E2 -8463.562} C_VEL
LIN {X 0,Y 452.515,Z 753.54,A -85,B 0,C 180,E1 -8464.454,E2 -8464.454} C_VEL
LIN {X 0,Y 452.658,Z 750.566,A -85,B 0,C 180,E1 -8465.792,E2 -8465.792} C_VEL
LIN {X 0,Y 452.728,Z 746.531,A -85,B 0,C 180,E1 -8467.134,E2 -8467.134} C_VEL
LIN {X 0,Y 452.977,Z 740.312,A -85,B 0,C 180,E1 -8468.701,E2 -8468.701} C_VEL
LIN {X 0,Y 453.291,Z 733.488,A -85,B 0,C 180,E1 -8470.045,E2 -8470.045} C_VEL
LIN {X 0,Y 453.748,Z 725.021,A -85,B 0,C 180,E1 -8471.39,E2 -8471.39} C_VEL
LIN {X 0,Y 454.103,Z 716.33,A -85,B 0,C 180,E1 -8472.514,E2 -8472.514} C_VEL
LIN {X 0,Y 454.596,Z 705.607,A -85,B 0,C 180,E1 -8473.637,E2 -8473.637} C_VEL
LIN {X 0,Y 455.205,Z 695.024,A -85,B 0,C 180,E1 -8474.53,E2 -8474.53} C_VEL
LIN {X 0,Y 455.657,Z 683.435,A -85,B 0,C 180,E1 -8475.315,E2 -8475.315} C_VEL
LIN {X 0,Y 456.129,Z 670.282,A -85,B 0,C 180,E1 -8475.987,E2 -8475.987} C_VEL
LIN {X 0,Y 456.476,Z 657.281,A -85,B 0,C 180,E1 -8476.462,E2 -8476.462} C_VEL
LIN {X 0,Y 456.754,Z 643.753,A -85,B 0,C 180,E1 -8476.768,E2 -8476.768} C_VEL
LIN {X 0,Y 457.909,Z 558.781,A -85,B 0,C 180,E1 -8478.304,E2 -8478.304} C_VEL
LIN {X 0,Y 455.04,Z 540.692,A -85,B 0,C 180,E1 -8478.779,E2 -8478.779} C_VEL
LIN {X 0,Y 456.015,Z 521.059,A -85,B 0,C 180,E1 -8482.057,E2 -8482.057} C_VEL
LIN {X 0,Y 457.247,Z 499.35,A -85,B 0,C 180,E1 -8485.735,E2 -8485.735} C_VEL
LIN {X 0,Y 457.06,Z 495.133,A -85,B 0,C 180,E1 -8486.482,E2 -8486.482} C_VEL
LIN {X 0,Y 453.876,Z 480.872,A -85,B 0,C 180,E1 -8489.193,E2 -8489.193} C_VEL
LIN {X 0,Y 453.511,Z 479.122,A -85,B 0,C 180,E1 -8489.538,E2 -8489.538} C_VEL
LIN {X 0,Y 453.493,Z 479.122,A -85,B 0,C 180,E1 -8493.189,E2 -8493.189} C_VEL
LIN {X 0,Y 453.457,Z 479.122,A -85,B 0,C 180,E1 -8496.299,E2 -8496.299} C_VEL
LIN {X 0,Y 453.519,Z 479.119,A -85,B 0,C 180,E1 -8499.447,E2 -8499.447} C_VEL
LIN {X 0,Y 453.465,Z 479.121,A -85,B 0,C 180,E1 -8502.995,E2 -8502.995} C_VEL
LIN {X 0,Y 453.466,Z 479.125,A -85,B 0,C 180,E1 -8505.779,E2 -8505.779} C_VEL
LIN {X 0,Y 453.481,Z 479.119,A -85,B 0,C 180,E1 -8508.209,E2 -8508.209} C_VEL
LIN {X 0,Y 453.489,Z 479.117,A -85,B 0,C 180,E1 -8510.794,E2 -8510.794} C_VEL
LIN {X 0,Y 453.456,Z 479.124,A -85,B 0,C 180,E1 -8513.917,E2 -8513.917} C_VEL
LIN {X 0,Y 453.485,Z 479.12,A -85,B 0,C 180,E1 -8517.151,E2 -8517.151} C_VEL
LIN {X 0,Y 453.477,Z 479.119,A -85,B 0,C 180,E1 -8520.268,E2 -8520.268} C_VEL
LIN {X 0,Y 453.509,Z 479.119,A -85,B 0,C 180,E1 -8523.294,E2 -8523.294} C_VEL
LIN {X 0,Y 453.521,Z 479.114,A -85,B 0,C 180,E1 -8524.117,E2 -8524.117} C_VEL
LIN {X 0,Y 452.857,Z 479.197,A -85,B 0,C 180,E1 -8524.858,E2 -8524.858} C_VEL
LIN {X 0,Y 449.959,Z 479.56,A -85,B 0,C 180,E1 -8526.061,E2 -8526.061} C_VEL
LIN {X 0,Y 447.519,Z 479.866,A -85,B 0,C 180,E1 -8527.032,E2 -8527.032} C_VEL
LIN {X 0,Y 446.5,Z 479.993,A -85,B 0,C 180,E1 -8527.782,E2 -8527.782} C_VEL
LIN {X 0,Y 446.433,Z 479.998,A -85,B 0,C 180,E1 -8528.036,E2 -8528.036} C_VEL
LIN {X 0,Y 446.477,Z 479.991,A -85,B 0,C 180,E1 -8530.815,E2 -8530.815} C_VEL
LIN {X 0,Y 446.498,Z 479.992,A -85,B 0,C 180,E1 -8533.772,E2 -8533.772} C_VEL
LIN {X 0,Y 446.517,Z 479.992,A -85,B 0,C 180,E1 -8537.384,E2 -8537.384} C_VEL
LIN {X 0,Y 446.541,Z 479.984,A -85,B 0,C 180,E1 -8540.945,E2 -8540.945} C_VEL
LIN {X 0,Y 446.649,Z 479.974,A -85,B 0,C 180,E1 -8543.676,E2 -8543.676} C_VEL
LIN {X 0,Y 446.711,Z 479.967,A -85,B 0,C 180,E1 -8547.295,E2 -8547.295} C_VEL
LIN {X 0,Y 446.796,Z 479.952,A -85,B 0,C 180,E1 -8550,E2 -8550} C_VEL
LIN {X 0,Y 446.712,Z 479.962,A -85,B 0,C 180,E1 -8552.705,E2 -8552.705} C_VEL
LIN {X 0,Y 446.641,Z 479.97,A -85,B 0,C 180,E1 -8556.324,E2 -8556.324} C_VEL
LIN {X 0,Y 446.54,Z 479.986,A -85,B 0,C 180,E1 -8559.055,E2 -8559.055} C_VEL
LIN {X 0,Y 446.523,Z 479.985,A -85,B 0,C 180,E1 -8562.73,E2 -8562.73} C_VEL
LIN {X 0,Y 446.498,Z 479.988,A -85,B 0,C 180,E1 -8566.228,E2 -8566.228} C_VEL
LIN {X 0,Y 446.471,Z 479.998,A -85,B 0,C 180,E1 -8569.303,E2 -8569.303} C_VEL
LIN {X 0,Y 446.42,Z 479.998,A -85,B 0,C 180,E1 -8572.2,E2 -8572.2} C_VEL
LIN {X 0,Y 446.46,Z 479.997,A -85,B 0,C 180,E1 -8575.152,E2 -8575.152} C_VEL
LIN {X 0,Y 446.486,Z 479.989,A -85,B 0,C 180,E1 -8578.179,E2 -8578.179} C_VEL
LIN {X 0,Y 446.421,Z 480,A -85,B 0,C 180,E1 -8581.775,E2 -8581.775} C_VEL
LIN {X 0,Y 446.43,Z 479.996,A -85,B 0,C 180,E1 -8584.523,E2 -8584.523} C_VEL
LIN {X 0,Y 446.417,Z 479.998,A -85,B 0,C 180,E1 -8588.079,E2 -8588.079} C_VEL
LIN {X 0,Y 446.43,Z 479.999,A -85,B 0,C 180,E1 -8590.918,E2 -8590.918} C_VEL
LIN {X 0,Y 446.425,Z 479.999,A -85,B 0,C 180,E1 -8593.843,E2 -8593.843} C_VEL
LIN {X 0,Y 446.401,Z 480,A -85,B 0,C 180,E1 -8596.403,E2 -8596.403} C_VEL
LIN {X 0,Y 446.429,Z 480.001,A -85,B 0,C 180,E1 -8599.083,E2 -8599.083} C_VEL
LIN {X 0,Y 446.411,Z 479.999,A -85,B 0,C 180,E1 -8602.121,E2 -8602.121} C_VEL
LIN {X 0,Y 446.432,Z 480.003,A -85,B 0,C 180,E1 -8605.477,E2 -8605.477} C_VEL
LIN {X 0,Y 446.418,Z 480.001,A -85,B 0,C 180,E1 -8608.7,E2 -8608.7} C_VEL
LIN {X 0,Y 446.478,Z 479.994,A -85,B 0,C 180,E1 -8611.824,E2 -8611.824} C_VEL
LIN {X 0,Y 449.666,Z 494.752,A -85,B 0,C 180,E1 -8614.321,E2 -8614.321} C_VEL
LIN {X 0,Y 450.023,Z 499.34,A -85,B 0,C 180,E1 -8615.061,E2 -8615.061} C_VEL
LIN {X 0,Y 449.21,Z 519.536,A -85,B 0,C 180,E1 -8618.187,E2 -8618.187} C_VEL
LIN {X 0,Y 448.434,Z 539.457,A -85,B 0,C 180,E1 -8621.26,E2 -8621.26} C_VEL
LIN {X 0,Y 448.195,Z 546.376,A -85,B 0,C 180,E1 -8622.326,E2 -8622.326} C_VEL
LIN {X 0,Y 450.726,Z 563.493,A -85,B 0,C 180,E1 -8622.75,E2 -8622.75} C_VEL
LIN {X 0,Y 449.5,Z 657.22,A -85,B 0,C 180,E1 -8624.469,E2 -8624.469} C_VEL
LIN {X 0,Y 449.134,Z 669.683,A -85,B 0,C 180,E1 -8624.863,E2 -8624.863} C_VEL
LIN {X 0,Y 448.665,Z 683.009,A -85,B 0,C 180,E1 -8625.485,E2 -8625.485} C_VEL
LIN {X 0,Y 448.17,Z 695.601,A -85,B 0,C 180,E1 -8626.28,E2 -8626.28} C_VEL
LIN {X 0,Y 447.704,Z 706.374,A -85,B 0,C 180,E1 -8627.154,E2 -8627.154} C_VEL
LIN {X 0,Y 447.18,Z 716.892,A -85,B 0,C 180,E1 -8628.211,E2 -8628.211} C_VEL
LIN {X 0,Y 446.734,Z 726.05,A -85,B 0,C 180,E1 -8629.348,E2 -8629.348} C_VEL
LIN {X 0,Y 446.259,Z 734.938,A -85,B 0,C 180,E1 -8630.71,E2 -8630.71} C_VEL
LIN {X 0,Y 445.921,Z 742.085,A -85,B 0,C 180,E1 -8632.073,E2 -8632.073} C_VEL
LIN {X 0,Y 445.726,Z 748.555,A -85,B 0,C 180,E1 -8633.663,E2 -8633.663} C_VEL
LIN {X 0,Y 445.532,Z 752.802,A -85,B 0,C 180,E1 -8635.023,E2 -8635.023} C_VEL
LIN {X 0,Y 445.482,Z 755.953,A -85,B 0,C 180,E1 -8636.382,E2 -8636.382} C_VEL
LIN {X 0,Y 445.46,Z 757.514,A -85,B 0,C 180,E1 -8637.287,E2 -8637.287} C_VEL
LIN {X 0,Y 445.379,Z 758.602,A -85,B 0,C 180,E1 -8638.191,E2 -8638.191} C_VEL
LIN {X 0,Y 445.341,Z 759.283,A -85,B 0,C 180,E1 -8639.096,E2 -8639.096} C_VEL
LIN {X 0,Y 445.342,Z 759.569,A -85,B 0,C 180,E1 -8640,E2 -8640} C_VEL
LIN {X 0,Y 445.341,Z 759.412,A -85,B 0,C 180,E1 -8640.904,E2 -8640.904} C_VEL
LIN {X 0,Y 445.379,Z 758.828,A -85,B 0,C 180,E1 -8641.809,E2 -8641.809} C_VEL
LIN {X 0,Y 445.461,Z 757.843,A -85,B 0,C 180,E1 -8642.713,E2 -8642.713} C_VEL
LIN {X 0,Y 445.499,Z 756.433,A -85,B 0,C 180,E1 -8643.618,E2 -8643.618} C_VEL
LIN {X 0,Y 445.528,Z 753.463,A -85,B 0,C 180,E1 -8644.977,E2 -8644.977} C_VEL
LIN {X 0,Y 445.746,Z 749.402,A -85,B 0,C 180,E1 -8646.337,E2 -8646.337} C_VEL
LIN {X 0,Y 445.95,Z 743.13,A -85,B 0,C 180,E1 -8647.926,E2 -8647.926} C_VEL
LIN {X 0,Y 446.335,Z 736.26,A -85,B 0,C 180,E1 -8649.288,E2 -8649.288} C_VEL
LIN {X 0,Y 446.763,Z 727.623,A -85,B 0,C 180,E1 -8650.652,E2 -8650.652} C_VEL
LIN {X 0,Y 447.294,Z 717.837,A -85,B 0,C 180,E1 -8651.901,E2 -8651.901} C_VEL
LIN {X 0,Y 447.85,Z 707.207,A -85,B 0,C 180,E1 -8652.983,E2 -8652.983} C_VEL
LIN {X 0,Y 448.395,Z 695.386,A -85,B 0,C 180,E1 -8653.945,E2 -8653.945} C_VEL
LIN {X 0,Y 448.802,Z 683.651,A -85,B 0,C 180,E1 -8654.684,E2 -8654.684} C_VEL
LIN {X 0,Y 449.349,Z 670.451,A -85,B 0,C 180,E1 -8655.304,E2 -8655.304} C_VEL
LIN {X 0,Y 449.676,Z 658.206,A -85,B 0,C 180,E1 -8655.699,E2 -8655.699} C_VEL
LIN {X 0,Y 451.217,Z 562.357,A -85,B 0,C 180,E1 -8657.568,E2 -8657.568} C_VEL
LIN {X 0,Y 448.69,Z 547.434,A -85,B 0,C 180,E1 -8658.019,E2 -8658.019} C_VEL
LIN {X 0,Y 449.445,Z 525.625,A -85,B 0,C 180,E1 -8661.319,E2 -8661.319} C_VEL
LIN {X 0,Y 450.329,Z 503.223,A -85,B 0,C 180,E1 -8664.675,E2 -8664.675} C_VEL
LIN {X 0,Y 450.313,Z 496.522,A -85,B 0,C 180,E1 -8665.681,E2 -8665.681} C_VEL
LIN {X 0,Y 447.902,Z 485.204,A -85,B 0,C 180,E1 -8667.573,E2 -8667.573} C_VEL
LIN {X 0,Y 446.471,Z 479.999,A -85,B 0,C 180,E1 -8668.48,E2 -8668.48} C_VEL
LIN {X 0,Y 446.422,Z 480.005,A -85,B 0,C 180,E1 -8671.775,E2 -8671.775} C_VEL
LIN {X 0,Y 446.431,Z 480.003,A -85,B 0,C 180,E1 -8674.523,E2 -8674.523} C_VEL
LIN {X 0,Y 446.418,Z 480.003,A -85,B 0,C 180,E1 -8678.079,E2 -8678.079} C_VEL
LIN {X 0,Y 446.429,Z 480.003,A -85,B 0,C 180,E1 -8680.918,E2 -8680.918} C_VEL
LIN {X 0,Y 446.404,Z 480.001,A -85,B 0,C 180,E1 -8683.846,E2 -8683.846} C_VEL
LIN {X 0,Y 446.423,Z 480.004,A -85,B 0,C 180,E1 -8686.4,E2 -8686.4} C_VEL
LIN {X 0,Y 446.453,Z 479.997,A -85,B 0,C 180,E1 -8689.803,E2 -8689.803} C_VEL
LIN {X 0,Y 446.43,Z 480.003,A -85,B 0,C 180,E1 -8692.123,E2 -8692.123} C_VEL
LIN {X 0,Y 446.432,Z 479.999,A -85,B 0,C 180,E1 -8695.477,E2 -8695.477} C_VEL
LIN {X 0,Y 446.433,Z 480.002,A -85,B 0,C 180,E1 -8698.701,E2 -8698.701} C_VEL
LIN {X 0,Y 446.498,Z 480.096,A -85,B 0,C 180,E1 -8701.539,E2 -8701.539} C_VEL
LIN {X 0,Y 450.32,Z 495.983,A -85,B 0,C 180,E1 -8704.298,E2 -8704.298} C_VEL
LIN {X 0,Y 451.256,Z 501.017,A -85,B 0,C 180,E1 -8705.133,E2 -8705.133} C_VEL
LIN {X 0,Y 449.811,Z 523.177,A -85,B 0,C 180,E1 -8708.459,E2 -8708.459} C_VEL
LIN {X 0,Y 449.666,Z 525.254,A -85,B 0,C 180,E1 -8708.767,E2 -8708.767} C_VEL
LIN {X 0,Y 452.729,Z 544.738,A -85,B 0,C 180,E1 -8709.265,E2 -8709.265} C_VEL
LIN {X 0,Y 450.903,Z 662.896,A -85,B 0,C 180,E1 -8711.366,E2 -8711.366} C_VEL
LIN {X 0,Y 450.421,Z 677.586,A -85,B 0,C 180,E1 -8711.816,E2 -8711.816} C_VEL
LIN {X 0,Y 449.948,Z 690.79,A -85,B 0,C 180,E1 -8712.399,E2 -8712.399} C_VEL
LIN {X 0,Y 449.341,Z 704.24,A -85,B 0,C 180,E1 -8713.181,E2 -8713.181} C_VEL
LIN {X 0,Y 448.566,Z 716.579,A -85,B 0,C 180,E1 -8714.087,E2 -8714.087} C_VEL
LIN {X 0,Y 447.958,Z 727.905,A -85,B 0,C 180,E1 -8715.113,E2 -8715.113} C_VEL
LIN {X 0,Y 447.227,Z 739.226,A -85,B 0,C 180,E1 -8716.366,E2 -8716.366} C_VEL
LIN {X 0,Y 446.768,Z 749.369,A -85,B 0,C 180,E1 -8717.739,E2 -8717.739} C_VEL
LIN {X 0,Y 446.272,Z 757.749,A -85,B 0,C 180,E1 -8719.107,E2 -8719.107} C_VEL
LIN {X 0,Y 445.893,Z 765.737,A -85,B 0,C 180,E1 -8720.703,E2 -8720.703} C_VEL
LIN {X 0,Y 445.613,Z 772.118,A -85,B 0,C 180,E1 -8722.296,E2 -8722.296} C_VEL
LIN {X 0,Y 445.482,Z 777.245,A -85,B 0,C 180,E1 -8723.939,E2 -8723.939} C_VEL
LIN {X 0,Y 445.396,Z 780.821,A -85,B 0,C 180,E1 -8725.475,E2 -8725.475} C_VEL
LIN {X 0,Y 445.429,Z 783.671,A -85,B 0,C 180,E1 -8727.287,E2 -8727.287} C_VEL
LIN {X 0,Y 445.338,Z 785.083,A -85,B 0,C 180,E1 -8729.096,E2 -8729.096} C_VEL
LIN {X 0,Y 445.338,Z 785.078,A -85,B 0,C 180,E1 -8730.904,E2 -8730.904} C_VEL
LIN {X 0,Y 445.429,Z 783.644,A -85,B 0,C 180,E1 -8732.713,E2 -8732.713} C_VEL
LIN {X 0,Y 445.397,Z 780.768,A -85,B 0,C 180,E1 -8734.525,E2 -8734.525} C_VEL
LIN {X 0,Y 445.529,Z 776.379,A -85,B 0,C 180,E1 -8736.34,E2 -8736.34} C_VEL
LIN {X 0,Y 445.609,Z 772.01,A -85,B 0,C 180,E1 -8737.704,E2 -8737.704} C_VEL
LIN {X 0,Y 445.885,Z 765.595,A -85,B 0,C 180,E1 -8739.298,E2 -8739.298} C_VEL
LIN {X 0,Y 446.275,Z 757.581,A -85,B 0,C 180,E1 -8740.893,E2 -8740.893} C_VEL
LIN {X 0,Y 446.723,Z 749.174,A -85,B 0,C 180,E1 -8742.262,E2 -8742.262} C_VEL
LIN {X 0,Y 447.269,Z 739.004,A -85,B 0,C 180,E1 -8743.633,E2 -8743.633} C_VEL
LIN {X 0,Y 447.878,Z 727.678,A -85,B 0,C 180,E1 -8744.889,E2 -8744.889} C_VEL
LIN {X 0,Y 448.576,Z 716.372,A -85,B 0,C 180,E1 -8745.913,E2 -8745.913} C_VEL
LIN {X 0,Y 449.303,Z 704.021,A -85,B 0,C 180,E1 -8746.821,E2 -8746.821} C_VEL
LIN {X 0,Y 449.9,Z 691.414,A -85,B 0,C 180,E1 -8747.56,E2 -8747.56} C_VEL
LIN {X 0,Y 450.423,Z 677.483,A -85,B 0,C 180,E1 -8748.184,E2 -8748.184} C_VEL
LIN {X 0,Y 450.958,Z 663.003,A -85,B 0,C 180,E1 -8748.632,E2 -8748.632} C_VEL
LIN {X 0,Y 453.001,Z 545.758,A -85,B 0,C 180,E1 -8750.82,E2 -8750.82} C_VEL
LIN {X 0,Y 451.17,Z 532.331,A -85,B 0,C 180,E1 -8751.198,E2 -8751.198} C_VEL
LIN {X 0,Y 450.071,Z 526.38,A -85,B 0,C 180,E1 -8751.391,E2 -8751.391} C_VEL
LIN {X 0,Y 451.865,Z 506.325,A -85,B 0,C 180,E1 -8754.586,E2 -8754.586} C_VEL
